LIN {X 0,Y 490.653,Z 372.898,A -85,B 0,C 180,E1 -6548.135,E2 -6548.135} C_VEL
LIN {X 0,Y 489.787,Z 400.79,A -85,B 0,C 180,E1 -6551.814,E2 -6551.814} C_VEL
LIN {X 0,Y 489.394,Z 415.444,A -85,B 0,C 180,E1 -6553.727,E2 -6553.727} C_VEL
LIN {X 0,Y 491.542,Z 434.875,A -85,B 0,C 180,E1 -6554.12,E2 -6554.12} C_VEL
LIN {X 0,Y 490.743,Z 525.863,A -85,B 0,C 180,E1 -6555.565,E2 -6555.565} C_VEL
LIN {X 0,Y 490.418,Z 538.788,A -85,B 0,C 180,E1 -6555.926,E2 -6555.926} C_VEL
LIN {X 0,Y 490.051,Z 550.862,A -85,B 0,C 180,E1 -6556.418,E2 -6556.418} C_VEL
LIN {X 0,Y 489.656,Z 562.336,A -85,B 0,C 180,E1 -6557.04,E2 -6557.04} C_VEL
LIN {X 0,Y 489.306,Z 574.419,A -85,B 0,C 180,E1 -6557.892,E2 -6557.892} C_VEL
LIN {X 0,Y 488.89,Z 584.844,A -85,B 0,C 180,E1 -6558.809,E2 -6558.809} C_VEL
LIN {X 0,Y 488.611,Z 594.472,A -85,B 0,C 180,E1 -6559.851,E2 -6559.851} C_VEL
LIN {X 0,Y 488.372,Z 603.748,A -85,B 0,C 180,E1 -6561.1,E2 -6561.1} C_VEL
LIN {X 0,Y 488.223,Z 611.226,A -85,B 0,C 180,E1 -6562.348,E2 -6562.348} C_VEL
LIN {X 0,Y 488.085,Z 617.817,A -85,B 0,C 180,E1 -6563.74,E2 -6563.74} C_VEL
LIN {X 0,Y 488.036,Z 622.557,A -85,B 0,C 180,E1 -6565.043,E2 -6565.043} C_VEL
LIN {X 0,Y 488.119,Z 624.938,A -85,B 0,C 180,E1 -6565.872,E2 -6565.872} C_VEL
LIN {X 0,Y 488.124,Z 626.864,A -85,B 0,C 180,E1 -6566.698,E2 -6566.698} C_VEL
LIN {X 0,Y 488.054,Z 628.303,A -85,B 0,C 180,E1 -6567.524,E2 -6567.524} C_VEL
LIN {X 0,Y 488.022,Z 629.312,A -85,B 0,C 180,E1 -6568.349,E2 -6568.349} C_VEL
LIN {X 0,Y 488.018,Z 629.915,A -85,B 0,C 180,E1 -6569.175,E2 -6569.175} C_VEL
LIN {X 0,Y 488.029,Z 630.112,A -85,B 0,C 180,E1 -6570,E2 -6570} C_VEL
LIN {X 0,Y 488.024,Z 629.858,A -85,B 0,C 180,E1 -6570.825,E2 -6570.825} C_VEL
LIN {X 0,Y 488.036,Z 629.184,A -85,B 0,C 180,E1 -6571.65,E2 -6571.65} C_VEL
LIN {X 0,Y 488.072,Z 628.103,A -85,B 0,C 180,E1 -6572.476,E2 -6572.476} C_VEL
LIN {X 0,Y 488.128,Z 626.599,A -85,B 0,C 180,E1 -6573.301,E2 -6573.301} C_VEL
LIN {X 0,Y 488.126,Z 623.454,A -85,B 0,C 180,E1 -6574.542,E2 -6574.542} C_VEL
LIN {X 0,Y 488.195,Z 618.077,A -85,B 0,C 180,E1 -6576.063,E2 -6576.063} C_VEL
LIN {X 0,Y 488.22,Z 611.62,A -85,B 0,C 180,E1 -6577.444,E2 -6577.444} C_VEL
LIN {X 0,Y 488.343,Z 604.254,A -85,B 0,C 180,E1 -6578.691,E2 -6578.691} C_VEL
LIN {X 0,Y 488.562,Z 595.04,A -85,B 0,C 180,E1 -6579.94,E2 -6579.94} C_VEL
LIN {X 0,Y 488.865,Z 585.619,A -85,B 0,C 180,E1 -6580.981,E2 -6580.981} C_VEL
LIN {X 0,Y 489.197,Z 574.668,A -85,B 0,C 180,E1 -6581.962,E2 -6581.962} C_VEL
LIN {X 0,Y 489.551,Z 563.67,A -85,B 0,C 180,E1 -6582.751,E2 -6582.751} C_VEL
LIN {X 0,Y 489.887,Z 551.761,A -85,B 0,C 180,E1 -6583.428,E2 -6583.428} C_VEL
LIN {X 0,Y 490.278,Z 538.993,A -85,B 0,C 180,E1 -6583.972,E2 -6583.972} C_VEL
LIN {X 0,Y 490.602,Z 525.693,A -85,B 0,C 180,E1 -6584.36,E2 -6584.36} C_VEL
LIN {X 0,Y 490.844,Z 499.198,A -85,B 0,C 180,E1 -6584.803,E2 -6584.803} C_VEL
LIN {X 0,Y 491.269,Z 432.405,A -85,B 0,C 180,E1 -6585.878,E2 -6585.878} C_VEL
LIN {X 0,Y 489.151,Z 412.344,A -85,B 0,C 180,E1 -6586.298,E2 -6586.298} C_VEL
LIN {X 0,Y 489.707,Z 390.705,A -85,B 0,C 180,E1 -6589.093,E2 -6589.093} C_VEL
LIN {X 0,Y 490.304,Z 367.801,A -85,B 0,C 180,E1 -6592.103,E2 -6592.103} C_VEL
LIN {X 0,Y 491.003,Z 346.439,A -85,B 0,C 180,E1 -6594.977,E2 -6594.977} C_VEL
LIN {X 0,Y 491.359,Z 333.411,A -85,B 0,C 180,E1 -6596.779,E2 -6596.779} C_VEL
LIN {X 0,Y 488.723,Z 320.611,A -85,B 0,C 180,E1 -6598.777,E2 -6598.777} C_VEL
LIN {X 0,Y 488.706,Z 320.614,A -85,B 0,C 180,E1 -6601.954,E2 -6601.954} C_VEL
LIN {X 0,Y 488.722,Z 320.608,A -85,B 0,C 180,E1 -6604.947,E2 -6604.947} C_VEL
LIN {X 0,Y 488.677,Z 320.616,A -85,B 0,C 180,E1 -6608.2,E2 -6608.2} C_VEL
LIN {X 0,Y 488.695,Z 320.615,A -85,B 0,C 180,E1 -6610.341,E2 -6610.341} C_VEL
LIN {X 0,Y 488.677,Z 320.614,A -85,B 0,C 180,E1 -6613.656,E2 -6613.656} C_VEL
LIN {X 0,Y 488.677,Z 320.615,A -85,B 0,C 180,E1 -6616.344,E2 -6616.344} C_VEL
LIN {X 0,Y 488.706,Z 320.61,A -85,B 0,C 180,E1 -6619.673,E2 -6619.673} C_VEL
LIN {X 0,Y 488.651,Z 320.613,A -85,B 0,C 180,E1 -6622.838,E2 -6622.838} C_VEL
LIN {X 0,Y 488.719,Z 320.61,A -85,B 0,C 180,E1 -6625.886,E2 -6625.886} C_VEL
LIN {X 0,Y 488.684,Z 320.61,A -85,B 0,C 180,E1 -6628.819,E2 -6628.819} C_VEL
LIN {X 0,Y 488.693,Z 320.614,A -85,B 0,C 180,E1 -6631.668,E2 -6631.668} C_VEL
LIN {X 0,Y 488.695,Z 320.61,A -85,B 0,C 180,E1 -6634.961,E2 -6634.961} C_VEL
LIN {X 0,Y 488.684,Z 320.614,A -85,B 0,C 180,E1 -6638.042,E2 -6638.042} C_VEL
LIN {X 0,Y 488.709,Z 320.608,A -85,B 0,C 180,E1 -6640.685,E2 -6640.685} C_VEL
LIN {X 0,Y 488.756,Z 320.605,A -85,B 0,C 180,E1 -6644.144,E2 -6644.144} C_VEL
LIN {X 0,Y 488.736,Z 320.61,A -85,B 0,C 180,E1 -6646.077,E2 -6646.077} C_VEL
LIN {X 0,Y 491.729,Z 329.522,A -85,B 0,C 180,E1 -6646.349,E2 -6646.349} C_VEL
LIN {X 0,Y 490.884,Z 411.162,A -85,B 0,C 180,E1 -6647.703,E2 -6647.703} C_VEL
LIN {X 0,Y 490.845,Z 424.387,A -85,B 0,C 180,E1 -6648.096,E2 -6648.096} C_VEL
LIN {X 0,Y 490.644,Z 436.99,A -85,B 0,C 180,E1 -6648.641,E2 -6648.641} C_VEL
LIN {X 0,Y 490.383,Z 449.309,A -85,B 0,C 180,E1 -6649.366,E2 -6649.366} C_VEL
LIN {X 0,Y 490.036,Z 460.307,A -85,B 0,C 180,E1 -6650.194,E2 -6650.194} C_VEL
LIN {X 0,Y 489.745,Z 470.169,A -85,B 0,C 180,E1 -6651.125,E2 -6651.125} C_VEL
LIN {X 0,Y 489.407,Z 479.39,A -85,B 0,C 180,E1 -6652.2,E2 -6652.2} C_VEL
LIN {X 0,Y 489.033,Z 487.732,A -85,B 0,C 180,E1 -6653.398,E2 -6653.398} C_VEL
LIN {X 0,Y 488.876,Z 494.611,A -85,B 0,C 180,E1 -6654.638,E2 -6654.638} C_VEL
LIN {X 0,Y 488.585,Z 500.097,A -85,B 0,C 180,E1 -6655.875,E2 -6655.875} C_VEL
LIN {X 0,Y 488.461,Z 504.372,A -85,B 0,C 180,E1 -6657.113,E2 -6657.113} C_VEL
LIN {X 0,Y 488.395,Z 507.572,A -85,B 0,C 180,E1 -6658.35,E2 -6658.35} C_VEL
LIN {X 0,Y 488.302,Z 509.151,A -85,B 0,C 180,E1 -6659.175,E2 -6659.175} C_VEL
LIN {X 0,Y 488.274,Z 510.323,A -85,B 0,C 180,E1 -6660,E2 -6660} C_VEL
LIN {X 0,Y 488.28,Z 511.074,A -85,B 0,C 180,E1 -6660.824,E2 -6660.824} C_VEL
LIN {X 0,Y 488.145,Z 511.418,A -85,B 0,C 180,E1 -6661.65,E2 -6661.65} C_VEL
LIN {X 0,Y 488.243,Z 510.907,A -85,B 0,C 180,E1 -6663.3,E2 -6663.3} C_VEL
LIN {X 0,Y 488.28,Z 510.038,A -85,B 0,C 180,E1 -6664.127,E2 -6664.127} C_VEL
LIN {X 0,Y 488.292,Z 508.754,A -85,B 0,C 180,E1 -6664.954,E2 -6664.954} C_VEL
LIN {X 0,Y 488.415,Z 506.04,A -85,B 0,C 180,E1 -6666.195,E2 -6666.195} C_VEL
LIN {X 0,Y 488.535,Z 502.302,A -85,B 0,C 180,E1 -6667.439,E2 -6667.439} C_VEL
LIN {X 0,Y 488.653,Z 497.43,A -85,B 0,C 180,E1 -6668.685,E2 -6668.685} C_VEL
LIN {X 0,Y 488.843,Z 491.265,A -85,B 0,C 180,E1 -6669.934,E2 -6669.934} C_VEL
LIN {X 0,Y 489.121,Z 483.572,A -85,B 0,C 180,E1 -6671.185,E2 -6671.185} C_VEL
LIN {X 0,Y 489.359,Z 475.615,A -85,B 0,C 180,E1 -6672.235,E2 -6672.235} C_VEL
LIN {X 0,Y 489.707,Z 465.965,A -85,B 0,C 180,E1 -6673.274,E2 -6673.274} C_VEL
LIN {X 0,Y 490.05,Z 455.168,A -85,B 0,C 180,E1 -6674.217,E2 -6674.217} C_VEL
LIN {X 0,Y 490.374,Z 444.676,A -85,B 0,C 180,E1 -6674.949,E2 -6674.949} C_VEL
LIN {X 0,Y 490.66,Z 432.035,A -85,B 0,C 180,E1 -6675.632,E2 -6675.632} C_VEL
LIN {X 0,Y 490.858,Z 418.426,A -85,B 0,C 180,E1 -6676.167,E2 -6676.167} C_VEL
LIN {X 0,Y 490.986,Z 405.659,A -85,B 0,C 180,E1 -6676.488,E2 -6676.488} C_VEL
LIN {X 0,Y 491.581,Z 329.224,A -85,B 0,C 180,E1 -6677.701,E2 -6677.701} C_VEL
LIN {X 0,Y 488.75,Z 320.604,A -85,B 0,C 180,E1 -6677.95,E2 -6677.95} C_VEL
LIN {X 0,Y 488.708,Z 320.609,A -85,B 0,C 180,E1 -6681.07,E2 -6681.07} C_VEL
LIN {X 0,Y 488.689,Z 320.608,A -85,B 0,C 180,E1 -6683.745,E2 -6683.745} C_VEL
LIN {X 0,Y 488.792,Z 320.599,A -85,B 0,C 180,E1 -6686.943,E2 -6686.943} C_VEL
LIN {X 0,Y 488.709,Z 320.61,A -85,B 0,C 180,E1 -6690.362,E2 -6690.362} C_VEL
LIN {X 0,Y 488.729,Z 320.603,A -85,B 0,C 180,E1 -6693.483,E2 -6693.483} C_VEL
LIN {X 0,Y 488.682,Z 320.613,A -85,B 0,C 180,E1 -6696.354,E2 -6696.354} C_VEL
LIN {X 0,Y 488.7,Z 320.607,A -85,B 0,C 180,E1 -6699.254,E2 -6699.254} C_VEL
LIN {X 0,Y 488.706,Z 320.606,A -85,B 0,C 180,E1 -6701.599,E2 -6701.599} C_VEL
LIN {X 0,Y 488.7,Z 320.61,A -85,B 0,C 180,E1 -6704.802,E2 -6704.802} C_VEL
LIN {X 0,Y 488.69,Z 320.608,A -85,B 0,C 180,E1 -6707.474,E2 -6707.474} C_VEL
LIN {X 0,Y 488.731,Z 320.603,A -85,B 0,C 180,E1 -6709.676,E2 -6709.676} C_VEL
LIN {X 0,Y 488.673,Z 320.613,A -85,B 0,C 180,E1 -6712.523,E2 -6712.523} C_VEL
LIN {X 0,Y 488.011,Z 320.695,A -85,B 0,C 180,E1 -6713.211,E2 -6713.211} C_VEL
LIN {X 0,Y 485.159,Z 321.054,A -85,B 0,C 180,E1 -6714.329,E2 -6714.329} C_VEL
LIN {X 0,Y 482.762,Z 321.348,A -85,B 0,C 180,E1 -6715.23,E2 -6715.23} C_VEL
LIN {X 0,Y 481.756,Z 321.474,A -85,B 0,C 180,E1 -6715.926,E2 -6715.926} C_VEL
LIN {X 0,Y 481.688,Z 321.484,A -85,B 0,C 180,E1 -6716.162,E2 -6716.162} C_VEL
LIN {X 0,Y 481.648,Z 321.485,A -85,B 0,C 180,E1 -6719.417,E2 -6719.417} C_VEL
LIN {X 0,Y 481.698,Z 321.484,A -85,B 0,C 180,E1 -6722.168,E2 -6722.168} C_VEL
LIN {X 0,Y 481.716,Z 321.478,A -85,B 0,C 180,E1 -6724.97,E2 -6724.97} C_VEL
LIN {X 0,Y 481.648,Z 321.487,A -85,B 0,C 180,E1 -6727.705,E2 -6727.705} C_VEL
LIN {X 0,Y 481.703,Z 321.484,A -85,B 0,C 180,E1 -6730.393,E2 -6730.393} C_VEL
LIN {X 0,Y 481.688,Z 321.481,A -85,B 0,C 180,E1 -6733.034,E2 -6733.034} C_VEL
LIN {X 0,Y 481.687,Z 321.483,A -85,B 0,C 180,E1 -6735.639,E2 -6735.639} C_VEL
LIN {X 0,Y 481.748,Z 321.48,A -85,B 0,C 180,E1 -6738.215,E2 -6738.215} C_VEL
LIN {X 0,Y 481.76,Z 321.474,A -85,B 0,C 180,E1 -6741.612,E2 -6741.612} C_VEL
LIN {X 0,Y 481.814,Z 321.471,A -85,B 0,C 180,E1 -6744.14,E2 -6744.14} C_VEL
LIN {X 0,Y 481.926,Z 321.453,A -85,B 0,C 180,E1 -6747.493,E2 -6747.493} C_VEL
LIN {X 0,Y 481.903,Z 321.454,A -85,B 0,C 180,E1 -6750.836,E2 -6750.836} C_VEL
LIN {X 0,Y 481.926,Z 321.453,A -85,B 0,C 180,E1 -6752.508,E2 -6752.508} C_VEL
LIN {X 0,Y 481.814,Z 321.469,A -85,B 0,C 180,E1 -6755.861,E2 -6755.861} C_VEL
LIN {X 0,Y 481.76,Z 321.474,A -85,B 0,C 180,E1 -6758.389,E2 -6758.389} C_VEL
LIN {X 0,Y 481.749,Z 321.477,A -85,B 0,C 180,E1 -6761.785,E2 -6761.785} C_VEL
LIN {X 0,Y 481.741,Z 321.475,A -85,B 0,C 180,E1 -6765.225,E2 -6765.225} C_VEL
LIN {X 0,Y 481.71,Z 321.478,A -85,B 0,C 180,E1 -6768.722,E2 -6768.722} C_VEL
LIN {X 0,Y 481.645,Z 321.489,A -85,B 0,C 180,E1 -6771.395,E2 -6771.395} C_VEL
LIN {X 0,Y 481.676,Z 321.486,A -85,B 0,C 180,E1 -6774.113,E2 -6774.113} C_VEL
LIN {X 0,Y 481.746,Z 321.475,A -85,B 0,C 180,E1 -6777.14,E2 -6777.14} C_VEL
LIN {X 0,Y 481.678,Z 321.487,A -85,B 0,C 180,E1 -6779.742,E2 -6779.742} C_VEL
LIN {X 0,Y 481.672,Z 321.483,A -85,B 0,C 180,E1 -6782.675,E2 -6782.675} C_VEL
LIN {X 0,Y 481.641,Z 321.492,A -85,B 0,C 180,E1 -6785.71,E2 -6785.71} C_VEL
LIN {X 0,Y 481.671,Z 321.483,A -85,B 0,C 180,E1 -6788.86,E2 -6788.86} C_VEL
LIN {X 0,Y 481.652,Z 321.49,A -85,B 0,C 180,E1 -6791.913,E2 -6791.913} C_VEL
LIN {X 0,Y 481.655,Z 321.485,A -85,B 0,C 180,E1 -6794.459,E2 -6794.459} C_VEL
LIN {X 0,Y 481.648,Z 321.49,A -85,B 0,C 180,E1 -6797.84,E2 -6797.84} C_VEL
LIN {X 0,Y 481.662,Z 321.484,A -85,B 0,C 180,E1 -6800.655,E2 -6800.655} C_VEL
LIN {X 0,Y 481.629,Z 321.492,A -85,B 0,C 180,E1 -6803.377,E2 -6803.377} C_VEL
LIN {X 0,Y 481.678,Z 321.482,A -85,B 0,C 180,E1 -6806.328,E2 -6806.328} C_VEL
LIN {X 0,Y 481.652,Z 321.49,A -85,B 0,C 180,E1 -6809.418,E2 -6809.418} C_VEL
LIN {X 0,Y 481.702,Z 321.48,A -85,B 0,C 180,E1 -6812.169,E2 -6812.169} C_VEL
LIN {X 0,Y 481.715,Z 321.48,A -85,B 0,C 180,E1 -6814.97,E2 -6814.97} C_VEL
LIN {X 0,Y 481.696,Z 321.483,A -85,B 0,C 180,E1 -6815.913,E2 -6815.913} C_VEL
LIN {X 0,Y 484.725,Z 330.592,A -85,B 0,C 180,E1 -6816.19,E2 -6816.19} C_VEL
LIN {X 0,Y 484.061,Z 408.884,A -85,B 0,C 180,E1 -6817.457,E2 -6817.457} C_VEL
LIN {X 0,Y 483.915,Z 421.637,A -85,B 0,C 180,E1 -6817.815,E2 -6817.815} C_VEL
LIN {X 0,Y 483.75,Z 433.868,A -85,B 0,C 180,E1 -6818.326,E2 -6818.326} C_VEL
LIN {X 0,Y 483.457,Z 446.293,A -85,B 0,C 180,E1 -6819.025,E2 -6819.025} C_VEL
LIN {X 0,Y 483.096,Z 456.914,A -85,B 0,C 180,E1 -6819.787,E2 -6819.787} C_VEL
LIN {X 0,Y 482.759,Z 467.753,A -85,B 0,C 180,E1 -6820.77,E2 -6820.77} C_VEL
LIN {X 0,Y 482.412,Z 476.559,A -85,B 0,C 180,E1 -6821.747,E2 -6821.747} C_VEL
LIN {X 0,Y 482.1,Z 484.622,A -85,B 0,C 180,E1 -6822.831,E2 -6822.831} C_VEL
LIN {X 0,Y 481.854,Z 491.253,A -85,B 0,C 180,E1 -6823.912,E2 -6823.912} C_VEL
LIN {X 0,Y 481.621,Z 497.7,A -85,B 0,C 180,E1 -6825.205,E2 -6825.205} C_VEL
LIN {X 0,Y 481.43,Z 502.757,A -85,B 0,C 180,E1 -6826.493,E2 -6826.493} C_VEL
LIN {X 0,Y 481.375,Z 507.213,A -85,B 0,C 180,E1 -6828.014,E2 -6828.014} C_VEL
LIN {X 0,Y 481.26,Z 509.417,A -85,B 0,C 180,E1 -6829.057,E2 -6829.057} C_VEL
LIN {X 0,Y 481.183,Z 510.736,A -85,B 0,C 180,E1 -6829.906,E2 -6829.906} C_VEL
LIN {X 0,Y 481.219,Z 511.633,A -85,B 0,C 180,E1 -6830.756,E2 -6830.756} C_VEL
LIN {X 0,Y 481.205,Z 512.089,A -85,B 0,C 180,E1 -6831.602,E2 -6831.602} C_VEL
LIN {X 0,Y 481.297,Z 511.861,A -85,B 0,C 180,E1 -6833.197,E2 -6833.197} C_VEL
LIN {X 0,Y 481.291,Z 511.047,A -85,B 0,C 180,E1 -6834.134,E2 -6834.134} C_VEL
LIN {X 0,Y 481.355,Z 509.867,A -85,B 0,C 180,E1 -6834.975,E2 -6834.975} C_VEL
LIN {X 0,Y 481.394,Z 507.324,A -85,B 0,C 180,E1 -6836.234,E2 -6836.234} C_VEL
LIN {X 0,Y 481.518,Z 503.762,A -85,B 0,C 180,E1 -6837.491,E2 -6837.491} C_VEL
LIN {X 0,Y 481.668,Z 499.092,A -85,B 0,C 180,E1 -6838.746,E2 -6838.746} C_VEL
LIN {X 0,Y 481.926,Z 493.165,A -85,B 0,C 180,E1 -6840,E2 -6840} C_VEL
LIN {X 0,Y 482.206,Z 485.737,A -85,B 0,C 180,E1 -6841.253,E2 -6841.253} C_VEL
LIN {X 0,Y 482.601,Z 476.463,A -85,B 0,C 180,E1 -6842.504,E2 -6842.504} C_VEL
LIN {X 0,Y 482.949,Z 466.853,A -85,B 0,C 180,E1 -6843.546,E2 -6843.546} C_VEL
LIN {X 0,Y 483.238,Z 456.096,A -85,B 0,C 180,E1 -6844.484,E2 -6844.484} C_VEL
LIN {X 0,Y 483.609,Z 445.598,A -85,B 0,C 180,E1 -6845.212,E2 -6845.212} C_VEL
LIN {X 0,Y 483.863,Z 434.096,A -85,B 0,C 180,E1 -6845.836,E2 -6845.836} C_VEL
LIN {X 0,Y 484.003,Z 420.929,A -85,B 0,C 180,E1 -6846.357,E2 -6846.357} C_VEL
LIN {X 0,Y 484.123,Z 407.732,A -85,B 0,C 180,E1 -6846.696,E2 -6846.696} C_VEL
LIN {X 0,Y 484.791,Z 330.376,A -85,B 0,C 180,E1 -6847.974,E2 -6847.974} C_VEL
LIN {X 0,Y 481.72,Z 321.482,A -85,B 0,C 180,E1 -6848.265,E2 -6848.265} C_VEL
LIN {X 0,Y 481.728,Z 321.479,A -85,B 0,C 180,E1 -6851.786,E2 -6851.786} C_VEL
LIN {X 0,Y 481.742,Z 321.476,A -85,B 0,C 180,E1 -6855.225,E2 -6855.225} C_VEL
LIN {X 0,Y 481.645,Z 321.493,A -85,B 0,C 180,E1 -6858.725,E2 -6858.725} C_VEL
LIN {X 0,Y 481.625,Z 321.491,A -85,B 0,C 180,E1 -6861.396,E2 -6861.396} C_VEL
LIN {X 0,Y 481.646,Z 321.492,A -85,B 0,C 180,E1 -6864.115,E2 -6864.115} C_VEL
LIN {X 0,Y 481.646,Z 321.487,A -85,B 0,C 180,E1 -6867.115,E2 -6867.115} C_VEL
LIN {X 0,Y 481.66,Z 321.487,A -85,B 0,C 180,E1 -6869.743,E2 -6869.743} C_VEL
LIN {X 0,Y 481.656,Z 321.486,A -85,B 0,C 180,E1 -6872.676,E2 -6872.676} C_VEL
LIN {X 0,Y 481.653,Z 321.483,A -85,B 0,C 180,E1 -6875.202,E2 -6875.202} C_VEL
LIN {X 0,Y 481.634,Z 321.491,A -85,B 0,C 180,E1 -6878.003,E2 -6878.003} C_VEL
LIN {X 0,Y 481.627,Z 321.486,A -85,B 0,C 180,E1 -6881.045,E2 -6881.045} C_VEL
LIN {X 0,Y 481.658,Z 321.485,A -85,B 0,C 180,E1 -6884.458,E2 -6884.458} C_VEL
LIN {X 0,Y 481.633,Z 321.495,A -85,B 0,C 180,E1 -6887.837,E2 -6887.837} C_VEL
LIN {X 0,Y 481.669,Z 321.485,A -85,B 0,C 180,E1 -6891.14,E2 -6891.14} C_VEL
LIN {X 0,Y 481.661,Z 321.485,A -85,B 0,C 180,E1 -6894.797,E2 -6894.797} C_VEL
LIN {X 0,Y 481.66,Z 321.489,A -85,B 0,C 180,E1 -6897.811,E2 -6897.811} C_VEL
LIN {X 0,Y 481.736,Z 321.634,A -85,B 0,C 180,E1 -6900.659,E2 -6900.659} C_VEL
LIN {X 0,Y 484.857,Z 335.891,A -85,B 0,C 180,E1 -6902.832,E2 -6902.832} C_VEL
LIN {X 0,Y 484.986,Z 340.7,A -85,B 0,C 180,E1 -6903.511,E2 -6903.511} C_VEL
LIN {X 0,Y 484.028,Z 364.108,A -85,B 0,C 180,E1 -6906.712,E2 -6906.712} C_VEL
LIN {X 0,Y 483.302,Z 383.679,A -85,B 0,C 180,E1 -6909.351,E2 -6909.351} C_VEL
LIN {X 0,Y 482.633,Z 404.958,A -85,B 0,C 180,E1 -6912.194,E2 -6912.194} C_VEL
LIN {X 0,Y 482.405,Z 415.085,A -85,B 0,C 180,E1 -6913.501,E2 -6913.501} C_VEL
LIN {X 0,Y 484.667,Z 435.54,A -85,B 0,C 180,E1 -6913.918,E2 -6913.918} C_VEL
LIN {X 0,Y 483.827,Z 525.311,A -85,B 0,C 180,E1 -6915.381,E2 -6915.381} C_VEL
LIN {X 0,Y 483.44,Z 538.896,A -85,B 0,C 180,E1 -6915.772,E2 -6915.772} C_VEL
LIN {X 0,Y 483.036,Z 551.808,A -85,B 0,C 180,E1 -6916.324,E2 -6916.324} C_VEL
LIN {X 0,Y 482.616,Z 562.838,A -85,B 0,C 180,E1 -6916.955,E2 -6916.955} C_VEL
LIN {X 0,Y 482.262,Z 574.328,A -85,B 0,C 180,E1 -6917.791,E2 -6917.791} C_VEL
LIN {X 0,Y 481.809,Z 584.929,A -85,B 0,C 180,E1 -6918.749,E2 -6918.749} C_VEL
LIN {X 0,Y 481.565,Z 593.523,A -85,B 0,C 180,E1 -6919.701,E2 -6919.701} C_VEL
LIN {X 0,Y 481.312,Z 602.832,A -85,B 0,C 180,E1 -6920.969,E2 -6920.969} C_VEL
LIN {X 0,Y 481.142,Z 610.331,A -85,B 0,C 180,E1 -6922.235,E2 -6922.235} C_VEL
LIN {X 0,Y 481.078,Z 615.98,A -85,B 0,C 180,E1 -6923.417,E2 -6923.417} C_VEL
LIN {X 0,Y 481.019,Z 620.328,A -85,B 0,C 180,E1 -6924.55,E2 -6924.55} C_VEL
LIN {X 0,Y 481.059,Z 624.088,A -85,B 0,C 180,E1 -6925.811,E2 -6925.811} C_VEL
LIN {X 0,Y 481.073,Z 626.018,A -85,B 0,C 180,E1 -6926.65,E2 -6926.65} C_VEL
LIN {X 0,Y 480.998,Z 627.46,A -85,B 0,C 180,E1 -6927.488,E2 -6927.488} C_VEL
LIN {X 0,Y 480.968,Z 628.467,A -85,B 0,C 180,E1 -6928.325,E2 -6928.325} C_VEL
LIN {X 0,Y 480.966,Z 629.069,A -85,B 0,C 180,E1 -6929.163,E2 -6929.163} C_VEL
LIN {X 0,Y 480.981,Z 629.262,A -85,B 0,C 180,E1 -6930,E2 -6930} C_VEL
LIN {X 0,Y 480.975,Z 628.997,A -85,B 0,C 180,E1 -6930.837,E2 -6930.837} C_VEL
LIN {X 0,Y 480.985,Z 628.313,A -85,B 0,C 180,E1 -6931.674,E2 -6931.674} C_VEL
LIN {X 0,Y 481.019,Z 627.222,A -85,B 0,C 180,E1 -6932.512,E2 -6932.512} C_VEL
LIN {X 0,Y 481.078,Z 624.745,A -85,B 0,C 180,E1 -6933.769,E2 -6933.769} C_VEL
LIN {X 0,Y 481.039,Z 621.208,A -85,B 0,C 180,E1 -6935.029,E2 -6935.029} C_VEL
LIN {X 0,Y 481.121,Z 616.306,A -85,B 0,C 180,E1 -6936.35,E2 -6936.35} C_VEL
LIN {X 0,Y 481.181,Z 609.489,A -85,B 0,C 180,E1 -6937.764,E2 -6937.764} C_VEL
LIN {X 0,Y 481.313,Z 601.779,A -85,B 0,C 180,E1 -6939.031,E2 -6939.031} C_VEL
LIN {X 0,Y 481.559,Z 592.216,A -85,B 0,C 180,E1 -6940.299,E2 -6940.299} C_VEL
LIN {X 0,Y 481.819,Z 582.279,A -85,B 0,C 180,E1 -6941.357,E2 -6941.357} C_VEL
LIN {X 0,Y 482.174,Z 571.65,A -85,B 0,C 180,E1 -6942.28,E2 -6942.28} C_VEL
LIN {X 0,Y 482.584,Z 560.752,A -85,B 0,C 180,E1 -6943.046,E2 -6943.046} C_VEL
LIN {X 0,Y 482.961,Z 548.243,A -85,B 0,C 180,E1 -6943.732,E2 -6943.732} C_VEL
LIN {X 0,Y 483.417,Z 534.462,A -85,B 0,C 180,E1 -6944.282,E2 -6944.282} C_VEL
LIN {X 0,Y 483.793,Z 521.74,A -85,B 0,C 180,E1 -6944.62,E2 -6944.62} C_VEL
LIN {X 0,Y 484.493,Z 433.696,A -85,B 0,C 180,E1 -6946.075,E2 -6946.075} C_VEL
LIN {X 0,Y 482.144,Z 411.17,A -85,B 0,C 180,E1 -6946.568,E2 -6946.568} C_VEL
LIN {X 0,Y 482.642,Z 390.052,A -85,B 0,C 180,E1 -6949.348,E2 -6949.348} C_VEL
LIN {X 0,Y 483.337,Z 368.644,A -85,B 0,C 180,E1 -6952.213,E2 -6952.213} C_VEL
LIN {X 0,Y 484.083,Z 347.416,A -85,B 0,C 180,E1 -6955.129,E2 -6955.129} C_VEL
LIN {X 0,Y 484.459,Z 334.635,A -85,B 0,C 180,E1 -6956.942,E2 -6956.942} C_VEL
LIN {X 0,Y 481.694,Z 321.486,A -85,B 0,C 180,E1 -6959.05,E2 -6959.05} C_VEL
LIN {X 0,Y 481.659,Z 321.493,A -85,B 0,C 180,E1 -6962.189,E2 -6962.189} C_VEL
LIN {X 0,Y 481.661,Z 321.486,A -85,B 0,C 180,E1 -6965.203,E2 -6965.203} C_VEL
LIN {X 0,Y 481.668,Z 321.487,A -85,B 0,C 180,E1 -6968.859,E2 -6968.859} C_VEL
LIN {X 0,Y 481.631,Z 321.495,A -85,B 0,C 180,E1 -6972.163,E2 -6972.163} C_VEL
LIN {X 0,Y 481.656,Z 321.487,A -85,B 0,C 180,E1 -6975.542,E2 -6975.542} C_VEL
LIN {X 0,Y 481.628,Z 321.489,A -85,B 0,C 180,E1 -6978.955,E2 -6978.955} C_VEL
LIN {X 0,Y 481.633,Z 321.492,A -85,B 0,C 180,E1 -6981.996,E2 -6981.996} C_VEL
LIN {X 0,Y 481.68,Z 321.483,A -85,B 0,C 180,E1 -6985.317,E2 -6985.317} C_VEL
LIN {X 0,Y 481.64,Z 321.49,A -85,B 0,C 180,E1 -6988.311,E2 -6988.311} C_VEL
LIN {X 0,Y 481.655,Z 321.487,A -85,B 0,C 180,E1 -6991.215,E2 -6991.215} C_VEL
LIN {X 0,Y 481.621,Z 321.495,A -85,B 0,C 180,E1 -6994.038,E2 -6994.038} C_VEL
LIN {X 0,Y 481.654,Z 321.488,A -85,B 0,C 180,E1 -6996.818,E2 -6996.818} C_VEL
LIN {X 0,Y 481.659,Z 321.492,A -85,B 0,C 180,E1 -6999.501,E2 -6999.501} C_VEL
LIN {X 0,Y 481.665,Z 321.487,A -85,B 0,C 180,E1 -7002.156,E2 -7002.156} C_VEL
LIN {X 0,Y 481.74,Z 321.48,A -85,B 0,C 180,E1 -7004.775,E2 -7004.775} C_VEL
LIN {X 0,Y 481.681,Z 321.49,A -85,B 0,C 180,E1 -7005.814,E2 -7005.814} C_VEL
LIN {X 0,Y 484.997,Z 331.124,A -85,B 0,C 180,E1 -7006.124,E2 -7006.124} C_VEL
LIN {X 0,Y 484.028,Z 411.924,A -85,B 0,C 180,E1 -7007.5,E2 -7007.5} C_VEL
LIN {X 0,Y 483.966,Z 425.906,A -85,B 0,C 180,E1 -7007.924,E2 -7007.924} C_VEL
LIN {X 0,Y 483.762,Z 438.322,A -85,B 0,C 180,E1 -7008.477,E2 -7008.477} C_VEL
LIN {X 0,Y 483.516,Z 450.549,A -85,B 0,C 180,E1 -7009.214,E2 -7009.214} C_VEL
LIN {X 0,Y 483.124,Z 461.485,A -85,B 0,C 180,E1 -7010.052,E2 -7010.052} C_VEL
LIN {X 0,Y 482.81,Z 471.288,A -85,B 0,C 180,E1 -7010.997,E2 -7010.997} C_VEL
LIN {X 0,Y 482.4,Z 481.13,A -85,B 0,C 180,E1 -7012.173,E2 -7012.173} C_VEL
LIN {X 0,Y 482.073,Z 488.785,A -85,B 0,C 180,E1 -7013.302,E2 -7013.302} C_VEL
LIN {X 0,Y 481.881,Z 495.639,A -85,B 0,C 180,E1 -7014.56,E2 -7014.56} C_VEL
LIN {X 0,Y 481.575,Z 501.101,A -85,B 0,C 180,E1 -7015.815,E2 -7015.815} C_VEL
LIN {X 0,Y 481.439,Z 505.35,A -85,B 0,C 180,E1 -7017.071,E2 -7017.071} C_VEL
LIN {X 0,Y 481.37,Z 508.522,A -85,B 0,C 180,E1 -7018.326,E2 -7018.326} C_VEL
LIN {X 0,Y 481.277,Z 510.086,A -85,B 0,C 180,E1 -7019.163,E2 -7019.163} C_VEL
LIN {X 0,Y 481.247,Z 511.242,A -85,B 0,C 180,E1 -7020,E2 -7020} C_VEL
LIN {X 0,Y 481.252,Z 511.965,A -85,B 0,C 180,E1 -7020.836,E2 -7020.836} C_VEL
LIN {X 0,Y 481.1,Z 512.292,A -85,B 0,C 180,E1 -7021.674,E2 -7021.674} C_VEL
LIN {X 0,Y 481.198,Z 511.739,A -85,B 0,C 180,E1 -7023.349,E2 -7023.349} C_VEL
LIN {X 0,Y 481.247,Z 510.834,A -85,B 0,C 180,E1 -7024.187,E2 -7024.187} C_VEL
LIN {X 0,Y 481.264,Z 509.523,A -85,B 0,C 180,E1 -7025.026,E2 -7025.026} C_VEL
LIN {X 0,Y 481.385,Z 506.761,A -85,B 0,C 180,E1 -7026.286,E2 -7026.286} C_VEL
LIN {X 0,Y 481.512,Z 502.968,A -85,B 0,C 180,E1 -7027.548,E2 -7027.548} C_VEL
LIN {X 0,Y 481.657,Z 498.032,A -85,B 0,C 180,E1 -7028.812,E2 -7028.812} C_VEL
LIN {X 0,Y 481.845,Z 491.8,A -85,B 0,C 180,E1 -7030.08,E2 -7030.08} C_VEL
LIN {X 0,Y 482.152,Z 484.004,A -85,B 0,C 180,E1 -7031.348,E2 -7031.348} C_VEL
LIN {X 0,Y 482.477,Z 474.449,A -85,B 0,C 180,E1 -7032.589,E2 -7032.589} C_VEL
LIN {X 0,Y 482.819,Z 463.975,A -85,B 0,C 180,E1 -7033.682,E2 -7033.682} C_VEL
LIN {X 0,Y 483.202,Z 452.363,A -85,B 0,C 180,E1 -7034.638,E2 -7034.638} C_VEL
LIN {X 0,Y 483.576,Z 440.934,A -85,B 0,C 180,E1 -7035.38,E2 -7035.38} C_VEL
LIN {X 0,Y 483.837,Z 429.194,A -85,B 0,C 180,E1 -7035.966,E2 -7035.966} C_VEL
LIN {X 0,Y 483.994,Z 415.59,A -85,B 0,C 180,E1 -7036.452,E2 -7036.452} C_VEL
LIN {X 0,Y 484.109,Z 402.044,A -85,B 0,C 180,E1 -7036.751,E2 -7036.751} C_VEL
LIN {X 0,Y 484.663,Z 330.407,A -85,B 0,C 180,E1 -7037.909,E2 -7037.909} C_VEL
LIN {X 0,Y 481.728,Z 321.48,A -85,B 0,C 180,E1 -7038.161,E2 -7038.161} C_VEL
LIN {X 0,Y 481.704,Z 321.483,A -85,B 0,C 180,E1 -7040.972,E2 -7040.972} C_VEL
LIN {X 0,Y 481.674,Z 321.484,A -85,B 0,C 180,E1 -7044.113,E2 -7044.113} C_VEL
LIN {X 0,Y 481.747,Z 321.475,A -85,B 0,C 180,E1 -7047.139,E2 -7047.139} C_VEL
LIN {X 0,Y 481.678,Z 321.482,A -85,B 0,C 180,E1 -7049.741,E2 -7049.741} C_VEL
LIN {X 0,Y 481.67,Z 321.49,A -85,B 0,C 180,E1 -7052.674,E2 -7052.674} C_VEL
LIN {X 0,Y 481.635,Z 321.487,A -85,B 0,C 180,E1 -7055.709,E2 -7055.709} C_VEL
LIN {X 0,Y 481.67,Z 321.486,A -85,B 0,C 180,E1 -7058.859,E2 -7058.859} C_VEL
LIN {X 0,Y 481.651,Z 321.486,A -85,B 0,C 180,E1 -7061.912,E2 -7061.912} C_VEL
LIN {X 0,Y 481.653,Z 321.491,A -85,B 0,C 180,E1 -7064.457,E2 -7064.457} C_VEL
LIN {X 0,Y 481.646,Z 321.487,A -85,B 0,C 180,E1 -7067.839,E2 -7067.839} C_VEL
LIN {X 0,Y 481.679,Z 321.486,A -85,B 0,C 180,E1 -7070.651,E2 -7070.651} C_VEL
LIN {X 0,Y 481.629,Z 321.488,A -85,B 0,C 180,E1 -7073.375,E2 -7073.375} C_VEL
LIN {X 0,Y 481.688,Z 321.484,A -85,B 0,C 180,E1 -7076.162,E2 -7076.162} C_VEL
LIN {X 0,Y 481.054,Z 321.57,A -85,B 0,C 180,E1 -7076.859,E2 -7076.859} C_VEL
LIN {X 0,Y 478.198,Z 321.927,A -85,B 0,C 180,E1 -7077.991,E2 -7077.991} C_VEL
LIN {X 0,Y 475.753,Z 322.227,A -85,B 0,C 180,E1 -7078.904,E2 -7078.904} C_VEL
LIN {X 0,Y 474.691,Z 322.355,A -85,B 0,C 180,E1 -7079.609,E2 -7079.609} C_VEL
LIN {X 0,Y 474.599,Z 322.365,A -85,B 0,C 180,E1 -7079.848,E2 -7079.848} C_VEL
LIN {X 0,Y 474.695,Z 322.355,A -85,B 0,C 180,E1 -7082.68,E2 -7082.68} C_VEL
LIN {X 0,Y 474.657,Z 322.357,A -85,B 0,C 180,E1 -7085.507,E2 -7085.507} C_VEL
LIN {X 0,Y 474.668,Z 322.355,A -85,B 0,C 180,E1 -7089.185,E2 -7089.185} C_VEL
LIN {X 0,Y 474.655,Z 322.359,A -85,B 0,C 180,E1 -7091.884,E2 -7091.884} C_VEL
LIN {X 0,Y 474.697,Z 322.355,A -85,B 0,C 180,E1 -7094.544,E2 -7094.544} C_VEL
LIN {X 0,Y 474.702,Z 322.355,A -85,B 0,C 180,E1 -7098.038,E2 -7098.038} C_VEL
LIN {X 0,Y 474.725,Z 322.349,A -85,B 0,C 180,E1 -7101.487,E2 -7101.487} C_VEL
LIN {X 0,Y 474.777,Z 322.347,A -85,B 0,C 180,E1 -7104.052,E2 -7104.052} C_VEL
LIN {X 0,Y 474.892,Z 322.329,A -85,B 0,C 180,E1 -7107.456,E2 -7107.456} C_VEL
LIN {X 0,Y 474.91,Z 322.33,A -85,B 0,C 180,E1 -7110,E2 -7110} C_VEL
LIN {X 0,Y 474.892,Z 322.329,A -85,B 0,C 180,E1 -7112.545,E2 -7112.545} C_VEL
LIN {X 0,Y 474.777,Z 322.347,A -85,B 0,C 180,E1 -7115.948,E2 -7115.948} C_VEL
LIN {X 0,Y 474.726,Z 322.35,A -85,B 0,C 180,E1 -7118.514,E2 -7118.514} C_VEL
LIN {X 0,Y 474.702,Z 322.357,A -85,B 0,C 180,E1 -7121.963,E2 -7121.963} C_VEL
LIN {X 0,Y 474.698,Z 322.354,A -85,B 0,C 180,E1 -7125.456,E2 -7125.456} C_VEL
LIN {X 0,Y 474.663,Z 322.356,A -85,B 0,C 180,E1 -7129.011,E2 -7129.011} C_VEL
LIN {X 0,Y 474.59,Z 322.369,A -85,B 0,C 180,E1 -7131.729,E2 -7131.729} C_VEL
LIN {X 0,Y 474.658,Z 322.357,A -85,B 0,C 180,E1 -7134.493,E2 -7134.493} C_VEL
LIN {X 0,Y 474.698,Z 322.354,A -85,B 0,C 180,E1 -7137.339,E2 -7137.339} C_VEL
LIN {X 0,Y 474.603,Z 322.363,A -85,B 0,C 180,E1 -7140.811,E2 -7140.811} C_VEL
LIN {X 0,Y 474.638,Z 322.364,A -85,B 0,C 180,E1 -7143.985,E2 -7143.985} C_VEL
LIN {X 0,Y 474.574,Z 322.368,A -85,B 0,C 180,E1 -7146.9,E2 -7146.9} C_VEL
LIN {X 0,Y 474.628,Z 322.365,A -85,B 0,C 180,E1 -7149.648,E2 -7149.648} C_VEL
LIN {X 0,Y 474.614,Z 322.363,A -85,B 0,C 180,E1 -7152.935,E2 -7152.935} C_VEL
LIN {X 0,Y 474.607,Z 322.367,A -85,B 0,C 180,E1 -7155.895,E2 -7155.895} C_VEL
LIN {X 0,Y 474.628,Z 322.363,A -85,B 0,C 180,E1 -7159.041,E2 -7159.041} C_VEL
LIN {X 0,Y 474.611,Z 322.368,A -85,B 0,C 180,E1 -7161.705,E2 -7161.705} C_VEL
LIN {X 0,Y 474.624,Z 322.361,A -85,B 0,C 180,E1 -7164.726,E2 -7164.726} C_VEL
LIN {X 0,Y 474.636,Z 322.363,A -85,B 0,C 180,E1 -7167.788,E2 -7167.788} C_VEL
LIN {X 0,Y 474.625,Z 322.363,A -85,B 0,C 180,E1 -7170.885,E2 -7170.885} C_VEL
LIN {X 0,Y 474.661,Z 322.36,A -85,B 0,C 180,E1 -7173.629,E2 -7173.629} C_VEL
LIN {X 0,Y 474.646,Z 322.363,A -85,B 0,C 180,E1 -7175.692,E2 -7175.692} C_VEL
LIN {X 0,Y 477.845,Z 331.959,A -85,B 0,C 180,E1 -7175.982,E2 -7175.982} C_VEL
LIN {X 0,Y 477.163,Z 410.39,A -85,B 0,C 180,E1 -7177.284,E2 -7177.284} C_VEL
LIN {X 0,Y 477.046,Z 422.813,A -85,B 0,C 180,E1 -7177.647,E2 -7177.647} C_VEL
LIN {X 0,Y 476.821,Z 435.905,A -85,B 0,C 180,E1 -7178.215,E2 -7178.215} C_VEL
LIN {X 0,Y 476.502,Z 448.176,A -85,B 0,C 180,E1 -7178.93,E2 -7178.93} C_VEL
LIN {X 0,Y 476.112,Z 459.837,A -85,B 0,C 180,E1 -7179.816,E2 -7179.816} C_VEL
LIN {X 0,Y 475.728,Z 470.304,A -85,B 0,C 180,E1 -7180.811,E2 -7180.811} C_VEL
LIN {X 0,Y 475.339,Z 479.662,A -85,B 0,C 180,E1 -7181.912,E2 -7181.912} C_VEL
LIN {X 0,Y 475,Z 488.679,A -85,B 0,C 180,E1 -7183.231,E2 -7183.231} C_VEL
LIN {X 0,Y 474.737,Z 495.84,A -85,B 0,C 180,E1 -7184.546,E2 -7184.546} C_VEL
LIN {X 0,Y 474.488,Z 501.491,A -85,B 0,C 180,E1 -7185.854,E2 -7185.854} C_VEL
LIN {X 0,Y 474.361,Z 505.882,A -85,B 0,C 180,E1 -7187.16,E2 -7187.16} C_VEL
LIN {X 0,Y 474.345,Z 508.189,A -85,B 0,C 180,E1 -7188.029,E2 -7188.029} C_VEL
LIN {X 0,Y 474.228,Z 510.016,A -85,B 0,C 180,E1 -7188.892,E2 -7188.892} C_VEL
LIN {X 0,Y 474.143,Z 511.397,A -85,B 0,C 180,E1 -7189.755,E2 -7189.755} C_VEL
LIN {X 0,Y 474.178,Z 512.364,A -85,B 0,C 180,E1 -7190.617,E2 -7190.617} C_VEL
LIN {X 0,Y 474.18,Z 512.902,A -85,B 0,C 180,E1 -7191.477,E2 -7191.477} C_VEL
LIN {X 0,Y 474.264,Z 512.734,A -85,B 0,C 180,E1 -7193.192,E2 -7193.192} C_VEL
LIN {X 0,Y 474.26,Z 512.057,A -85,B 0,C 180,E1 -7194.046,E2 -7194.046} C_VEL
LIN {X 0,Y 474.305,Z 510.927,A -85,B 0,C 180,E1 -7194.9,E2 -7194.9} C_VEL
LIN {X 0,Y 474.303,Z 509.408,A -85,B 0,C 180,E1 -7195.752,E2 -7195.752} C_VEL
LIN {X 0,Y 474.416,Z 506.293,A -85,B 0,C 180,E1 -7197.028,E2 -7197.028} C_VEL
LIN {X 0,Y 474.574,Z 502.117,A -85,B 0,C 180,E1 -7198.303,E2 -7198.303} C_VEL
LIN {X 0,Y 474.817,Z 496.756,A -85,B 0,C 180,E1 -7199.576,E2 -7199.576} C_VEL
LIN {X 0,Y 475.146,Z 489.988,A -85,B 0,C 180,E1 -7200.848,E2 -7200.848} C_VEL
LIN {X 0,Y 475.513,Z 481.565,A -85,B 0,C 180,E1 -7202.118,E2 -7202.118} C_VEL
LIN {X 0,Y 475.89,Z 472.919,A -85,B 0,C 180,E1 -7203.175,E2 -7203.175} C_VEL
LIN {X 0,Y 476.272,Z 463.355,A -85,B 0,C 180,E1 -7204.126,E2 -7204.126} C_VEL
LIN {X 0,Y 476.544,Z 452.883,A -85,B 0,C 180,E1 -7204.971,E2 -7204.971} C_VEL
LIN {X 0,Y 476.93,Z 441.262,A -85,B 0,C 180,E1 -7205.709,E2 -7205.709} C_VEL
LIN {X 0,Y 477.06,Z 429.199,A -85,B 0,C 180,E1 -7206.291,E2 -7206.291} C_VEL
LIN {X 0,Y 477.221,Z 415.862,A -85,B 0,C 180,E1 -7206.74,E2 -7206.74} C_VEL
LIN {X 0,Y 477.302,Z 401.245,A -85,B 0,C 180,E1 -7207.031,E2 -7207.031} C_VEL
LIN {X 0,Y 478.193,Z 332.453,A -85,B 0,C 180,E1 -7208.193,E2 -7208.193} C_VEL
LIN {X 0,Y 474.712,Z 322.574,A -85,B 0,C 180,E1 -7208.514,E2 -7208.514} C_VEL
LIN {X 0,Y 474.674,Z 322.362,A -85,B 0,C 180,E1 -7208.729,E2 -7208.729} C_VEL
LIN {X 0,Y 474.693,Z 322.359,A -85,B 0,C 180,E1 -7212.269,E2 -7212.269} C_VEL
LIN {X 0,Y 474.684,Z 322.356,A -85,B 0,C 180,E1 -7215.767,E2 -7215.767} C_VEL
LIN {X 0,Y 474.598,Z 322.369,A -85,B 0,C 180,E1 -7219.013,E2 -7219.013} C_VEL
LIN {X 0,Y 474.574,Z 322.371,A -85,B 0,C 180,E1 -7221.73,E2 -7221.73} C_VEL
LIN {X 0,Y 474.625,Z 322.367,A -85,B 0,C 180,E1 -7224.495,E2 -7224.495} C_VEL
LIN {X 0,Y 474.597,Z 322.365,A -85,B 0,C 180,E1 -7227.327,E2 -7227.327} C_VEL
LIN {X 0,Y 474.591,Z 322.37,A -85,B 0,C 180,E1 -7230.232,E2 -7230.232} C_VEL
LIN {X 0,Y 474.619,Z 322.361,A -85,B 0,C 180,E1 -7233.222,E2 -7233.222} C_VEL
LIN {X 0,Y 474.574,Z 322.369,A -85,B 0,C 180,E1 -7236.325,E2 -7236.325} C_VEL
LIN {X 0,Y 474.605,Z 322.365,A -85,B 0,C 180,E1 -7239.644,E2 -7239.644} C_VEL
LIN {X 0,Y 474.573,Z 322.365,A -85,B 0,C 180,E1 -7242.939,E2 -7242.939} C_VEL
LIN {X 0,Y 474.606,Z 322.368,A -85,B 0,C 180,E1 -7245.894,E2 -7245.894} C_VEL
LIN {X 0,Y 474.609,Z 322.363,A -85,B 0,C 180,E1 -7249.044,E2 -7249.044} C_VEL
LIN {X 0,Y 474.609,Z 322.368,A -85,B 0,C 180,E1 -7251.705,E2 -7251.705} C_VEL
LIN {X 0,Y 474.623,Z 322.361,A -85,B 0,C 180,E1 -7254.725,E2 -7254.725} C_VEL
LIN {X 0,Y 474.639,Z 322.364,A -85,B 0,C 180,E1 -7257.788,E2 -7257.788} C_VEL
LIN {X 0,Y 474.666,Z 322.422,A -85,B 0,C 180,E1 -7260.416,E2 -7260.416} C_VEL
LIN {X 0,Y 478.094,Z 338.449,A -85,B 0,C 180,E1 -7262.89,E2 -7262.89} C_VEL
LIN {X 0,Y 477.652,Z 351.673,A -85,B 0,C 180,E1 -7264.742,E2 -7264.742} C_VEL
LIN {X 0,Y 476.593,Z 377.996,A -85,B 0,C 180,E1 -7268.367,E2 -7268.367} C_VEL
LIN {X 0,Y 475.728,Z 402.575,A -85,B 0,C 180,E1 -7271.704,E2 -7271.704} C_VEL
LIN {X 0,Y 475.38,Z 414.058,A -85,B 0,C 180,E1 -7273.25,E2 -7273.25} C_VEL
LIN {X 0,Y 477.804,Z 436.037,A -85,B 0,C 180,E1 -7273.711,E2 -7273.711} C_VEL
LIN {X 0,Y 476.92,Z 524.691,A -85,B 0,C 180,E1 -7275.192,E2 -7275.192} C_VEL
LIN {X 0,Y 476.485,Z 538.185,A -85,B 0,C 180,E1 -7275.587,E2 -7275.587} C_VEL
LIN {X 0,Y 476.061,Z 550.545,A -85,B 0,C 180,E1 -7276.119,E2 -7276.119} C_VEL
LIN {X 0,Y 475.575,Z 563.273,A -85,B 0,C 180,E1 -7276.867,E2 -7276.867} C_VEL
LIN {X 0,Y 475.216,Z 574.177,A -85,B 0,C 180,E1 -7277.685,E2 -7277.685} C_VEL
LIN {X 0,Y 474.786,Z 583.887,A -85,B 0,C 180,E1 -7278.581,E2 -7278.581} C_VEL
LIN {X 0,Y 474.536,Z 592.53,A -85,B 0,C 180,E1 -7279.547,E2 -7279.547} C_VEL
LIN {X 0,Y 474.244,Z 601.886,A -85,B 0,C 180,E1 -7280.833,E2 -7280.833} C_VEL
LIN {X 0,Y 474.059,Z 609.415,A -85,B 0,C 180,E1 -7282.118,E2 -7282.118} C_VEL
LIN {X 0,Y 474.001,Z 615.53,A -85,B 0,C 180,E1 -7283.42,E2 -7283.42} C_VEL
LIN {X 0,Y 473.901,Z 620.838,A -85,B 0,C 180,E1 -7284.895,E2 -7284.895} C_VEL
LIN {X 0,Y 474,Z 623.232,A -85,B 0,C 180,E1 -7285.748,E2 -7285.748} C_VEL
LIN {X 0,Y 474.024,Z 625.167,A -85,B 0,C 180,E1 -7286.6,E2 -7286.6} C_VEL
LIN {X 0,Y 473.942,Z 626.613,A -85,B 0,C 180,E1 -7287.45,E2 -7287.45} C_VEL
LIN {X 0,Y 473.914,Z 627.621,A -85,B 0,C 180,E1 -7288.3,E2 -7288.3} C_VEL
LIN {X 0,Y 473.915,Z 628.221,A -85,B 0,C 180,E1 -7289.15,E2 -7289.15} C_VEL
LIN {X 0,Y 473.932,Z 628.411,A -85,B 0,C 180,E1 -7290,E2 -7290} C_VEL
LIN {X 0,Y 473.925,Z 628.138,A -85,B 0,C 180,E1 -7290.85,E2 -7290.85} C_VEL
LIN {X 0,Y 473.933,Z 627.447,A -85,B 0,C 180,E1 -7291.699,E2 -7291.699} C_VEL
LIN {X 0,Y 473.965,Z 626.344,A -85,B 0,C 180,E1 -7292.549,E2 -7292.549} C_VEL
LIN {X 0,Y 474.035,Z 623.849,A -85,B 0,C 180,E1 -7293.825,E2 -7293.825} C_VEL
LIN {X 0,Y 473.969,Z 620.283,A -85,B 0,C 180,E1 -7295.104,E2 -7295.104} C_VEL
LIN {X 0,Y 474.056,Z 615.703,A -85,B 0,C 180,E1 -7296.357,E2 -7296.357} C_VEL
LIN {X 0,Y 474.082,Z 609.625,A -85,B 0,C 180,E1 -7297.667,E2 -7297.667} C_VEL
LIN {X 0,Y 474.208,Z 602.165,A -85,B 0,C 180,E1 -7298.952,E2 -7298.952} C_VEL
LIN {X 0,Y 474.445,Z 592.863,A -85,B 0,C 180,E1 -7300.239,E2 -7300.239} C_VEL
LIN {X 0,Y 474.68,Z 583.33,A -85,B 0,C 180,E1 -7301.313,E2 -7301.313} C_VEL
LIN {X 0,Y 475.122,Z 573.645,A -85,B 0,C 180,E1 -7302.209,E2 -7302.209} C_VEL
LIN {X 0,Y 475.505,Z 562.796,A -85,B 0,C 180,E1 -7303.026,E2 -7303.026} C_VEL
LIN {X 0,Y 475.931,Z 550.185,A -85,B 0,C 180,E1 -7303.775,E2 -7303.775} C_VEL
LIN {X 0,Y 476.408,Z 536.957,A -85,B 0,C 180,E1 -7304.36,E2 -7304.36} C_VEL
LIN {X 0,Y 476.796,Z 523.769,A -85,B 0,C 180,E1 -7304.757,E2 -7304.757} C_VEL
LIN {X 0,Y 477.129,Z 494.735,A -85,B 0,C 180,E1 -7305.266,E2 -7305.266} C_VEL
LIN {X 0,Y 477.594,Z 433.824,A -85,B 0,C 180,E1 -7306.308,E2 -7306.308} C_VEL
LIN {X 0,Y 475.128,Z 410.026,A -85,B 0,C 180,E1 -7306.848,E2 -7306.848} C_VEL
LIN {X 0,Y 475.689,Z 389.232,A -85,B 0,C 180,E1 -7309.64,E2 -7309.64} C_VEL
LIN {X 0,Y 476.371,Z 369.562,A -85,B 0,C 180,E1 -7312.327,E2 -7312.327} C_VEL
LIN {X 0,Y 477.19,Z 348.48,A -85,B 0,C 180,E1 -7315.284,E2 -7315.284} C_VEL
LIN {X 0,Y 477.655,Z 337.243,A -85,B 0,C 180,E1 -7316.9,E2 -7316.9} C_VEL
LIN {X 0,Y 475.856,Z 327.651,A -85,B 0,C 180,E1 -7318.444,E2 -7318.444} C_VEL
LIN {X 0,Y 474.654,Z 322.363,A -85,B 0,C 180,E1 -7319.371,E2 -7319.371} C_VEL
LIN {X 0,Y 474.617,Z 322.37,A -85,B 0,C 180,E1 -7322.43,E2 -7322.43} C_VEL
LIN {X 0,Y 474.613,Z 322.365,A -85,B 0,C 180,E1 -7325.468,E2 -7325.468} C_VEL
LIN {X 0,Y 474.61,Z 322.369,A -85,B 0,C 180,E1 -7328.458,E2 -7328.458} C_VEL
LIN {X 0,Y 474.606,Z 322.368,A -85,B 0,C 180,E1 -7331.787,E2 -7331.787} C_VEL
LIN {X 0,Y 474.618,Z 322.364,A -85,B 0,C 180,E1 -7334.702,E2 -7334.702} C_VEL
LIN {X 0,Y 474.587,Z 322.37,A -85,B 0,C 180,E1 -7337.769,E2 -7337.769} C_VEL
LIN {X 0,Y 474.62,Z 322.364,A -85,B 0,C 180,E1 -7340.451,E2 -7340.451} C_VEL
LIN {X 0,Y 474.572,Z 322.37,A -85,B 0,C 180,E1 -7343.675,E2 -7343.675} C_VEL
LIN {X 0,Y 474.617,Z 322.361,A -85,B 0,C 180,E1 -7346.777,E2 -7346.777} C_VEL
LIN {X 0,Y 474.589,Z 322.371,A -85,B 0,C 180,E1 -7349.768,E2 -7349.768} C_VEL
LIN {X 0,Y 474.603,Z 322.364,A -85,B 0,C 180,E1 -7352.684,E2 -7352.684} C_VEL
LIN {X 0,Y 474.623,Z 322.368,A -85,B 0,C 180,E1 -7355.505,E2 -7355.505} C_VEL
LIN {X 0,Y 474.64,Z 322.364,A -85,B 0,C 180,E1 -7359.184,E2 -7359.184} C_VEL
LIN {X 0,Y 474.621,Z 322.367,A -85,B 0,C 180,E1 -7361.883,E2 -7361.883} C_VEL
LIN {X 0,Y 474.699,Z 322.356,A -85,B 0,C 180,E1 -7364.544,E2 -7364.544} C_VEL
LIN {X 0,Y 474.655,Z 322.365,A -85,B 0,C 180,E1 -7365.532,E2 -7365.532} C_VEL
LIN {X 0,Y 478.123,Z 332.101,A -85,B 0,C 180,E1 -7365.867,E2 -7365.867} C_VEL
LIN {X 0,Y 477.181,Z 414.011,A -85,B 0,C 180,E1 -7367.317,E2 -7367.317} C_VEL
LIN {X 0,Y 477.144,Z 426.874,A -85,B 0,C 180,E1 -7367.722,E2 -7367.722} C_VEL
LIN {X 0,Y 476.923,Z 438.786,A -85,B 0,C 180,E1 -7368.255,E2 -7368.255} C_VEL
LIN {X 0,Y 476.696,Z 450.32,A -85,B 0,C 180,E1 -7368.95,E2 -7368.95} C_VEL
LIN {X 0,Y 476.288,Z 461.459,A -85,B 0,C 180,E1 -7369.801,E2 -7369.801} C_VEL
LIN {X 0,Y 475.953,Z 471.484,A -85,B 0,C 180,E1 -7370.759,E2 -7370.759} C_VEL
LIN {X 0,Y 475.569,Z 480.009,A -85,B 0,C 180,E1 -7371.758,E2 -7371.758} C_VEL
LIN {X 0,Y 475.197,Z 488.692,A -85,B 0,C 180,E1 -7373.014,E2 -7373.014} C_VEL
LIN {X 0,Y 475.027,Z 495.647,A -85,B 0,C 180,E1 -7374.268,E2 -7374.268} C_VEL
LIN {X 0,Y 474.706,Z 500.446,A -85,B 0,C 180,E1 -7375.329,E2 -7375.329} C_VEL
LIN {X 0,Y 474.44,Z 505.069,A -85,B 0,C 180,E1 -7376.603,E2 -7376.603} C_VEL
LIN {X 0,Y 474.288,Z 507.544,A -85,B 0,C 180,E1 -7377.452,E2 -7377.452} C_VEL
LIN {X 0,Y 474.346,Z 509.484,A -85,B 0,C 180,E1 -7378.302,E2 -7378.302} C_VEL
LIN {X 0,Y 474.252,Z 511.032,A -85,B 0,C 180,E1 -7379.15,E2 -7379.15} C_VEL
LIN {X 0,Y 474.22,Z 512.171,A -85,B 0,C 180,E1 -7380,E2 -7380} C_VEL
LIN {X 0,Y 474.223,Z 512.864,A -85,B 0,C 180,E1 -7380.849,E2 -7380.849} C_VEL
LIN {X 0,Y 474.055,Z 513.173,A -85,B 0,C 180,E1 -7381.699,E2 -7381.699} C_VEL
LIN {X 0,Y 474.086,Z 513.068,A -85,B 0,C 180,E1 -7382.549,E2 -7382.549} C_VEL
LIN {X 0,Y 474.153,Z 512.568,A -85,B 0,C 180,E1 -7383.399,E2 -7383.399} C_VEL
LIN {X 0,Y 474.215,Z 511.627,A -85,B 0,C 180,E1 -7384.249,E2 -7384.249} C_VEL
LIN {X 0,Y 474.238,Z 510.288,A -85,B 0,C 180,E1 -7385.101,E2 -7385.101} C_VEL
LIN {X 0,Y 474.36,Z 507.472,A -85,B 0,C 180,E1 -7386.379,E2 -7386.379} C_VEL
LIN {X 0,Y 474.484,Z 503.62,A -85,B 0,C 180,E1 -7387.66,E2 -7387.66} C_VEL
LIN {X 0,Y 474.666,Z 498.612,A -85,B 0,C 180,E1 -7388.943,E2 -7388.943} C_VEL
LIN {X 0,Y 474.868,Z 492.301,A -85,B 0,C 180,E1 -7390.229,E2 -7390.229} C_VEL
LIN {X 0,Y 475.184,Z 484.382,A -85,B 0,C 180,E1 -7391.517,E2 -7391.517} C_VEL
LIN {X 0,Y 475.522,Z 475.175,A -85,B 0,C 180,E1 -7392.721,E2 -7392.721} C_VEL
LIN {X 0,Y 475.878,Z 465.234,A -85,B 0,C 180,E1 -7393.776,E2 -7393.776} C_VEL
LIN {X 0,Y 476.244,Z 455.168,A -85,B 0,C 180,E1 -7394.638,E2 -7394.638} C_VEL
LIN {X 0,Y 476.591,Z 444.205,A -85,B 0,C 180,E1 -7395.392,E2 -7395.392} C_VEL
LIN {X 0,Y 476.889,Z 432.118,A -85,B 0,C 180,E1 -7396.04,E2 -7396.04} C_VEL
LIN {X 0,Y 477.068,Z 419.323,A -85,B 0,C 180,E1 -7396.542,E2 -7396.542} C_VEL
LIN {X 0,Y 477.21,Z 406.471,A -85,B 0,C 180,E1 -7396.869,E2 -7396.869} C_VEL
LIN {X 0,Y 477.754,Z 331.673,A -85,B 0,C 180,E1 -7398.114,E2 -7398.114} C_VEL
LIN {X 0,Y 474.67,Z 322.361,A -85,B 0,C 180,E1 -7398.399,E2 -7398.399} C_VEL
LIN {X 0,Y 474.636,Z 322.361,A -85,B 0,C 180,E1 -7401.116,E2 -7401.116} C_VEL
LIN {X 0,Y 474.656,Z 322.361,A -85,B 0,C 180,E1 -7404.493,E2 -7404.493} C_VEL
LIN {X 0,Y 474.682,Z 322.354,A -85,B 0,C 180,E1 -7407.334,E2 -7407.334} C_VEL
LIN {X 0,Y 474.604,Z 322.365,A -85,B 0,C 180,E1 -7410.23,E2 -7410.23} C_VEL
LIN {X 0,Y 474.624,Z 322.361,A -85,B 0,C 180,E1 -7413.221,E2 -7413.221} C_VEL
LIN {X 0,Y 474.588,Z 322.368,A -85,B 0,C 180,E1 -7416.323,E2 -7416.323} C_VEL
LIN {X 0,Y 474.617,Z 322.361,A -85,B 0,C 180,E1 -7419.646,E2 -7419.646} C_VEL
LIN {X 0,Y 474.613,Z 322.364,A -85,B 0,C 180,E1 -7422.934,E2 -7422.934} C_VEL
LIN {X 0,Y 474.604,Z 322.365,A -85,B 0,C 180,E1 -7425.894,E2 -7425.894} C_VEL
LIN {X 0,Y 474.626,Z 322.361,A -85,B 0,C 180,E1 -7429.04,E2 -7429.04} C_VEL
LIN {X 0,Y 474.609,Z 322.363,A -85,B 0,C 180,E1 -7431.704,E2 -7431.704} C_VEL
LIN {X 0,Y 474.628,Z 322.363,A -85,B 0,C 180,E1 -7434.726,E2 -7434.726} C_VEL
LIN {X 0,Y 474.634,Z 322.361,A -85,B 0,C 180,E1 -7437.788,E2 -7437.788} C_VEL
LIN {X 0,Y 474.599,Z 322.365,A -85,B 0,C 180,E1 -7439.848,E2 -7439.848} C_VEL
LIN {X 0,Y 473.924,Z 322.452,A -85,B 0,C 180,E1 -7440.557,E2 -7440.557} C_VEL
LIN {X 0,Y 471.092,Z 322.802,A -85,B 0,C 180,E1 -7441.709,E2 -7441.709} C_VEL
LIN {X 0,Y 468.704,Z 323.102,A -85,B 0,C 180,E1 -7442.638,E2 -7442.638} C_VEL
LIN {X 0,Y 467.679,Z 323.226,A -85,B 0,C 180,E1 -7443.355,E2 -7443.355} C_VEL
LIN {X 0,Y 467.595,Z 323.236,A -85,B 0,C 180,E1 -7443.598,E2 -7443.598} C_VEL
LIN {X 0,Y 467.59,Z 323.242,A -85,B 0,C 180,E1 -7446.468,E2 -7446.468} C_VEL
LIN {X 0,Y 467.62,Z 323.235,A -85,B 0,C 180,E1 -7449.777,E2 -7449.777} C_VEL
LIN {X 0,Y 467.606,Z 323.239,A -85,B 0,C 180,E1 -7452.507,E2 -7452.507} C_VEL
LIN {X 0,Y 467.604,Z 323.235,A -85,B 0,C 180,E1 -7455.196,E2 -7455.196} C_VEL
LIN {X 0,Y 467.653,Z 323.232,A -85,B 0,C 180,E1 -7457.855,E2 -7457.855} C_VEL
LIN {X 0,Y 467.679,Z 323.226,A -85,B 0,C 180,E1 -7461.357,E2 -7461.357} C_VEL
LIN {X 0,Y 467.741,Z 323.222,A -85,B 0,C 180,E1 -7463.963,E2 -7463.963} C_VEL
LIN {X 0,Y 467.858,Z 323.205,A -85,B 0,C 180,E1 -7467.417,E2 -7467.417} C_VEL
LIN {X 0,Y 467.881,Z 323.206,A -85,B 0,C 180,E1 -7470,E2 -7470} C_VEL
LIN {X 0,Y 467.857,Z 323.205,A -85,B 0,C 180,E1 -7472.583,E2 -7472.583} C_VEL
LIN {X 0,Y 467.741,Z 323.224,A -85,B 0,C 180,E1 -7476.038,E2 -7476.038} C_VEL
LIN {X 0,Y 467.679,Z 323.227,A -85,B 0,C 180,E1 -7478.643,E2 -7478.643} C_VEL
LIN {X 0,Y 467.654,Z 323.234,A -85,B 0,C 180,E1 -7482.146,E2 -7482.146} C_VEL
LIN {X 0,Y 467.637,Z 323.234,A -85,B 0,C 180,E1 -7485.695,E2 -7485.695} C_VEL
LIN {X 0,Y 467.616,Z 323.234,A -85,B 0,C 180,E1 -7488.765,E2 -7488.765} C_VEL
LIN {X 0,Y 467.579,Z 323.24,A -85,B 0,C 180,E1 -7491.269,E2 -7491.269} C_VEL
LIN {X 0,Y 467.573,Z 323.245,A -85,B 0,C 180,E1 -7493.944,E2 -7493.944} C_VEL
LIN {X 0,Y 467.615,Z 323.234,A -85,B 0,C 180,E1 -7496.801,E2 -7496.801} C_VEL
LIN {X 0,Y 467.553,Z 323.246,A -85,B 0,C 180,E1 -7499.739,E2 -7499.739} C_VEL
LIN {X 0,Y 467.582,Z 323.238,A -85,B 0,C 180,E1 -7502.759,E2 -7502.759} C_VEL
LIN {X 0,Y 467.556,Z 323.247,A -85,B 0,C 180,E1 -7505.89,E2 -7505.89} C_VEL
LIN {X 0,Y 467.582,Z 323.24,A -85,B 0,C 180,E1 -7509.145,E2 -7509.145} C_VEL
LIN {X 0,Y 467.586,Z 323.238,A -85,B 0,C 180,E1 -7512.568,E2 -7512.568} C_VEL
LIN {X 0,Y 467.566,Z 323.242,A -85,B 0,C 180,E1 -7515.053,E2 -7515.053} C_VEL
LIN {X 0,Y 467.589,Z 323.241,A -85,B 0,C 180,E1 -7517.441,E2 -7517.441} C_VEL
LIN {X 0,Y 467.561,Z 323.242,A -85,B 0,C 180,E1 -7520.854,E2 -7520.854} C_VEL
LIN {X 0,Y 467.56,Z 323.242,A -85,B 0,C 180,E1 -7524.262,E2 -7524.262} C_VEL
LIN {X 0,Y 467.581,Z 323.242,A -85,B 0,C 180,E1 -7527.322,E2 -7527.322} C_VEL
LIN {X 0,Y 467.571,Z 323.24,A -85,B 0,C 180,E1 -7530.668,E2 -7530.668} C_VEL
LIN {X 0,Y 467.618,Z 323.238,A -85,B 0,C 180,E1 -7533.2,E2 -7533.2} C_VEL
LIN {X 0,Y 467.668,Z 323.412,A -85,B 0,C 180,E1 -7535.491,E2 -7535.491} C_VEL
LIN {X 0,Y 470.98,Z 333.354,A -85,B 0,C 180,E1 -7535.778,E2 -7535.778} C_VEL
LIN {X 0,Y 470.293,Z 411.573,A -85,B 0,C 180,E1 -7537.108,E2 -7537.108} C_VEL
LIN {X 0,Y 470.146,Z 423.059,A -85,B 0,C 180,E1 -7537.448,E2 -7537.448} C_VEL
LIN {X 0,Y 469.948,Z 435.898,A -85,B 0,C 180,E1 -7538.004,E2 -7538.004} C_VEL
LIN {X 0,Y 469.616,Z 448.214,A -85,B 0,C 180,E1 -7538.721,E2 -7538.721} C_VEL
LIN {X 0,Y 469.254,Z 458.784,A -85,B 0,C 180,E1 -7539.508,E2 -7539.508} C_VEL
LIN {X 0,Y 468.85,Z 469.578,A -85,B 0,C 180,E1 -7540.518,E2 -7540.518} C_VEL
LIN {X 0,Y 468.423,Z 479.278,A -85,B 0,C 180,E1 -7541.635,E2 -7541.635} C_VEL
LIN {X 0,Y 468.117,Z 487.167,A -85,B 0,C 180,E1 -7542.752,E2 -7542.752} C_VEL
LIN {X 0,Y 467.781,Z 494.661,A -85,B 0,C 180,E1 -7544.061,E2 -7544.061} C_VEL
LIN {X 0,Y 467.551,Z 499.953,A -85,B 0,C 180,E1 -7545.195,E2 -7545.195} C_VEL
LIN {X 0,Y 467.379,Z 504.904,A -85,B 0,C 180,E1 -7546.522,E2 -7546.522} C_VEL
LIN {X 0,Y 467.299,Z 508.667,A -85,B 0,C 180,E1 -7547.846,E2 -7547.846} C_VEL
LIN {X 0,Y 467.209,Z 510.603,A -85,B 0,C 180,E1 -7548.723,E2 -7548.723} C_VEL
LIN {X 0,Y 467.106,Z 512.049,A -85,B 0,C 180,E1 -7549.599,E2 -7549.599} C_VEL
LIN {X 0,Y 467.12,Z 513.076,A -85,B 0,C 180,E1 -7550.474,E2 -7550.474} C_VEL
LIN {X 0,Y 467.134,Z 513.71,A -85,B 0,C 180,E1 -7551.347,E2 -7551.347} C_VEL
LIN {X 0,Y 467.145,Z 513.89,A -85,B 0,C 180,E1 -7552.219,E2 -7552.219} C_VEL
LIN {X 0,Y 467.227,Z 513.65,A -85,B 0,C 180,E1 -7553.11,E2 -7553.11} C_VEL
LIN {X 0,Y 467.232,Z 513.053,A -85,B 0,C 180,E1 -7553.956,E2 -7553.956} C_VEL
LIN {X 0,Y 467.275,Z 512.01,A -85,B 0,C 180,E1 -7554.823,E2 -7554.823} C_VEL
LIN {X 0,Y 467.27,Z 510.546,A -85,B 0,C 180,E1 -7555.688,E2 -7555.688} C_VEL
LIN {X 0,Y 467.389,Z 507.535,A -85,B 0,C 180,E1 -7556.984,E2 -7556.984} C_VEL
LIN {X 0,Y 467.56,Z 503.464,A -85,B 0,C 180,E1 -7558.278,E2 -7558.278} C_VEL
LIN {X 0,Y 467.816,Z 498.211,A -85,B 0,C 180,E1 -7559.57,E2 -7559.57} C_VEL
LIN {X 0,Y 468.19,Z 491.606,A -85,B 0,C 180,E1 -7560.861,E2 -7560.861} C_VEL
LIN {X 0,Y 468.568,Z 483.323,A -85,B 0,C 180,E1 -7562.149,E2 -7562.149} C_VEL
LIN {X 0,Y 468.952,Z 474.838,A -85,B 0,C 180,E1 -7563.222,E2 -7563.222} C_VEL
LIN {X 0,Y 469.305,Z 465.551,A -85,B 0,C 180,E1 -7564.187,E2 -7564.187} C_VEL
LIN {X 0,Y 469.643,Z 455.362,A -85,B 0,C 180,E1 -7565.044,E2 -7565.044} C_VEL
LIN {X 0,Y 469.984,Z 444.165,A -85,B 0,C 180,E1 -7565.794,E2 -7565.794} C_VEL
LIN {X 0,Y 470.24,Z 431.679,A -85,B 0,C 180,E1 -7566.436,E2 -7566.436} C_VEL
LIN {X 0,Y 470.394,Z 419.102,A -85,B 0,C 180,E1 -7566.892,E2 -7566.892} C_VEL
LIN {X 0,Y 470.483,Z 406.314,A -85,B 0,C 180,E1 -7567.187,E2 -7567.187} C_VEL
LIN {X 0,Y 471.38,Z 333.514,A -85,B 0,C 180,E1 -7568.453,E2 -7568.453} C_VEL
LIN {X 0,Y 467.635,Z 323.24,A -85,B 0,C 180,E1 -7568.815,E2 -7568.815} C_VEL
LIN {X 0,Y 467.647,Z 323.237,A -85,B 0,C 180,E1 -7572.351,E2 -7572.351} C_VEL
LIN {X 0,Y 467.628,Z 323.236,A -85,B 0,C 180,E1 -7575.874,E2 -7575.874} C_VEL
LIN {X 0,Y 467.544,Z 323.247,A -85,B 0,C 180,E1 -7579.312,E2 -7579.312} C_VEL
LIN {X 0,Y 467.523,Z 323.253,A -85,B 0,C 180,E1 -7582.075,E2 -7582.075} C_VEL
LIN {X 0,Y 467.554,Z 323.244,A -85,B 0,C 180,E1 -7584.891,E2 -7584.891} C_VEL
LIN {X 0,Y 467.545,Z 323.246,A -85,B 0,C 180,E1 -7587.774,E2 -7587.774} C_VEL
LIN {X 0,Y 467.547,Z 323.243,A -85,B 0,C 180,E1 -7591.04,E2 -7591.04} C_VEL
LIN {X 0,Y 467.579,Z 323.242,A -85,B 0,C 180,E1 -7594.24,E2 -7594.24} C_VEL
LIN {X 0,Y 467.52,Z 323.244,A -85,B 0,C 180,E1 -7597.181,E2 -7597.181} C_VEL
LIN {X 0,Y 467.56,Z 323.242,A -85,B 0,C 180,E1 -7600.267,E2 -7600.267} C_VEL
LIN {X 0,Y 467.548,Z 323.247,A -85,B 0,C 180,E1 -7603.746,E2 -7603.746} C_VEL
LIN {X 0,Y 467.55,Z 323.245,A -85,B 0,C 180,E1 -7606.254,E2 -7606.254} C_VEL
LIN {X 0,Y 467.563,Z 323.246,A -85,B 0,C 180,E1 -7609.733,E2 -7609.733} C_VEL
LIN {X 0,Y 467.545,Z 323.243,A -85,B 0,C 180,E1 -7612.815,E2 -7612.815} C_VEL
LIN {X 0,Y 467.58,Z 323.244,A -85,B 0,C 180,E1 -7615.76,E2 -7615.76} C_VEL
LIN {X 0,Y 467.572,Z 323.242,A -85,B 0,C 180,E1 -7618.955,E2 -7618.955} C_VEL
LIN {X 0,Y 467.659,Z 323.418,A -85,B 0,C 180,E1 -7620.207,E2 -7620.207} C_VEL
LIN {X 0,Y 471.094,Z 339.293,A -85,B 0,C 180,E1 -7622.694,E2 -7622.694} C_VEL
LIN {X 0,Y 471.055,Z 345.848,A -85,B 0,C 180,E1 -7623.637,E2 -7623.637} C_VEL
LIN {X 0,Y 469.977,Z 368.99,A -85,B 0,C 180,E1 -7626.887,E2 -7626.887} C_VEL
LIN {X 0,Y 469.125,Z 390.314,A -85,B 0,C 180,E1 -7629.844,E2 -7629.844} C_VEL
LIN {X 0,Y 468.403,Z 411.554,A -85,B 0,C 180,E1 -7632.763,E2 -7632.763} C_VEL
LIN {X 0,Y 468.353,Z 413.362,A -85,B 0,C 180,E1 -7633.01,E2 -7633.01} C_VEL
LIN {X 0,Y 470.925,Z 436.072,A -85,B 0,C 180,E1 -7633.497,E2 -7633.497} C_VEL
LIN {X 0,Y 470.008,Z 523.776,A -85,B 0,C 180,E1 -7634.997,E2 -7634.997} C_VEL
LIN {X 0,Y 469.546,Z 537.287,A -85,B 0,C 180,E1 -7635.397,E2 -7635.397} C_VEL
LIN {X 0,Y 469.082,Z 550.196,A -85,B 0,C 180,E1 -7635.964,E2 -7635.964} C_VEL
LIN {X 0,Y 468.546,Z 562.019,A -85,B 0,C 180,E1 -7636.666,E2 -7636.666} C_VEL
LIN {X 0,Y 468.176,Z 573.247,A -85,B 0,C 180,E1 -7637.517,E2 -7637.517} C_VEL
LIN {X 0,Y 467.766,Z 582.802,A -85,B 0,C 180,E1 -7638.407,E2 -7638.407} C_VEL
LIN {X 0,Y 467.511,Z 591.506,A -85,B 0,C 180,E1 -7639.388,E2 -7639.388} C_VEL
LIN {X 0,Y 467.193,Z 599.518,A -85,B 0,C 180,E1 -7640.475,E2 -7640.475} C_VEL
LIN {X 0,Y 467.002,Z 607.339,A -85,B 0,C 180,E1 -7641.78,E2 -7641.78} C_VEL
LIN {X 0,Y 466.915,Z 613.619,A -85,B 0,C 180,E1 -7643.084,E2 -7643.084} C_VEL
LIN {X 0,Y 466.894,Z 618.579,A -85,B 0,C 180,E1 -7644.385,E2 -7644.385} C_VEL
LIN {X 0,Y 466.94,Z 622.367,A -85,B 0,C 180,E1 -7645.684,E2 -7645.684} C_VEL
LIN {X 0,Y 466.976,Z 624.31,A -85,B 0,C 180,E1 -7646.549,E2 -7646.549} C_VEL
LIN {X 0,Y 466.887,Z 625.762,A -85,B 0,C 180,E1 -7647.412,E2 -7647.412} C_VEL
LIN {X 0,Y 466.861,Z 626.771,A -85,B 0,C 180,E1 -7648.275,E2 -7648.275} C_VEL
LIN {X 0,Y 466.864,Z 627.369,A -85,B 0,C 180,E1 -7649.137,E2 -7649.137} C_VEL
LIN {X 0,Y 466.884,Z 627.557,A -85,B 0,C 180,E1 -7650,E2 -7650} C_VEL
LIN {X 0,Y 466.875,Z 627.279,A -85,B 0,C 180,E1 -7650.862,E2 -7650.862} C_VEL
LIN {X 0,Y 466.881,Z 626.578,A -85,B 0,C 180,E1 -7651.725,E2 -7651.725} C_VEL
LIN {X 0,Y 466.911,Z 625.467,A -85,B 0,C 180,E1 -7652.588,E2 -7652.588} C_VEL
LIN {X 0,Y 466.992,Z 622.956,A -85,B 0,C 180,E1 -7653.883,E2 -7653.883} C_VEL
LIN {X 0,Y 466.9,Z 619.366,A -85,B 0,C 180,E1 -7655.182,E2 -7655.182} C_VEL
LIN {X 0,Y 466.982,Z 614.011,A -85,B 0,C 180,E1 -7656.639,E2 -7656.639} C_VEL
LIN {X 0,Y 467.042,Z 607.51,A -85,B 0,C 180,E1 -7658.001,E2 -7658.001} C_VEL
LIN {X 0,Y 467.182,Z 599.721,A -85,B 0,C 180,E1 -7659.306,E2 -7659.306} C_VEL
LIN {X 0,Y 467.471,Z 590.088,A -85,B 0,C 180,E1 -7660.613,E2 -7660.613} C_VEL
LIN {X 0,Y 467.829,Z 580.093,A -85,B 0,C 180,E1 -7661.701,E2 -7661.701} C_VEL
LIN {X 0,Y 468.208,Z 568.513,A -85,B 0,C 180,E1 -7662.723,E2 -7662.723} C_VEL
LIN {X 0,Y 468.669,Z 556.647,A -85,B 0,C 180,E1 -7663.551,E2 -7663.551} C_VEL
LIN {X 0,Y 469.259,Z 543.534,A -85,B 0,C 180,E1 -7664.252,E2 -7664.252} C_VEL
LIN {X 0,Y 469.681,Z 530.352,A -85,B 0,C 180,E1 -7664.764,E2 -7664.764} C_VEL
LIN {X 0,Y 470.042,Z 516.286,A -85,B 0,C 180,E1 -7665.113,E2 -7665.113} C_VEL
LIN {X 0,Y 470.874,Z 435.203,A -85,B 0,C 180,E1 -7666.525,E2 -7666.525} C_VEL
LIN {X 0,Y 468.164,Z 408.943,A -85,B 0,C 180,E1 -7667.135,E2 -7667.135} C_VEL
LIN {X 0,Y 468.699,Z 388.431,A -85,B 0,C 180,E1 -7669.946,E2 -7669.946} C_VEL
LIN {X 0,Y 469.452,Z 368.875,A -85,B 0,C 180,E1 -7672.674,E2 -7672.674} C_VEL
LIN {X 0,Y 470.321,Z 349.557,A -85,B 0,C 180,E1 -7675.443,E2 -7675.443} C_VEL
LIN {X 0,Y 470.785,Z 338.443,A -85,B 0,C 180,E1 -7677.085,E2 -7677.085} C_VEL
LIN {X 0,Y 468.639,Z 327.727,A -85,B 0,C 180,E1 -7678.87,E2 -7678.87} C_VEL
LIN {X 0,Y 467.624,Z 323.239,A -85,B 0,C 180,E1 -7679.675,E2 -7679.675} C_VEL
LIN {X 0,Y 467.582,Z 323.246,A -85,B 0,C 180,E1 -7682.759,E2 -7682.759} C_VEL
LIN {X 0,Y 467.553,Z 323.246,A -85,B 0,C 180,E1 -7685.89,E2 -7685.89} C_VEL
LIN {X 0,Y 467.554,Z 323.244,A -85,B 0,C 180,E1 -7689.148,E2 -7689.148} C_VEL
LIN {X 0,Y 467.567,Z 323.243,A -85,B 0,C 180,E1 -7691.404,E2 -7691.404} C_VEL
LIN {X 0,Y 467.568,Z 323.241,A -85,B 0,C 180,E1 -7695.052,E2 -7695.052} C_VEL
LIN {X 0,Y 467.564,Z 323.242,A -85,B 0,C 180,E1 -7698.725,E2 -7698.725} C_VEL
LIN {X 0,Y 467.543,Z 323.247,A -85,B 0,C 180,E1 -7701.953,E2 -7701.953} C_VEL
LIN {X 0,Y 467.552,Z 323.242,A -85,B 0,C 180,E1 -7705.166,E2 -7705.166} C_VEL
LIN {X 0,Y 467.559,Z 323.245,A -85,B 0,C 180,E1 -7708.258,E2 -7708.258} C_VEL
LIN {X 0,Y 467.541,Z 323.246,A -85,B 0,C 180,E1 -7711.248,E2 -7711.248} C_VEL
LIN {X 0,Y 467.563,Z 323.243,A -85,B 0,C 180,E1 -7714.405,E2 -7714.405} C_VEL
LIN {X 0,Y 467.553,Z 323.245,A -85,B 0,C 180,E1 -7716.994,E2 -7716.994} C_VEL
LIN {X 0,Y 467.589,Z 323.242,A -85,B 0,C 180,E1 -7719.775,E2 -7719.775} C_VEL
LIN {X 0,Y 467.578,Z 323.241,A -85,B 0,C 180,E1 -7722.505,E2 -7722.505} C_VEL
LIN {X 0,Y 467.616,Z 323.243,A -85,B 0,C 180,E1 -7725.235,E2 -7725.235} C_VEL
LIN {X 0,Y 471.438,Z 333.757,A -85,B 0,C 180,E1 -7725.616,E2 -7725.616} C_VEL
LIN {X 0,Y 470.371,Z 414.23,A -85,B 0,C 180,E1 -7727.076,E2 -7727.076} C_VEL
LIN {X 0,Y 470.342,Z 427.993,A -85,B 0,C 180,E1 -7727.514,E2 -7727.514} C_VEL
LIN {X 0,Y 470.098,Z 439.327,A -85,B 0,C 180,E1 -7728.028,E2 -7728.028} C_VEL
LIN {X 0,Y 469.883,Z 450.179,A -85,B 0,C 180,E1 -7728.678,E2 -7728.678} C_VEL
LIN {X 0,Y 469.471,Z 461.499,A -85,B 0,C 180,E1 -7729.542,E2 -7729.542} C_VEL
LIN {X 0,Y 469.111,Z 471.695,A -85,B 0,C 180,E1 -7730.514,E2 -7730.514} C_VEL
LIN {X 0,Y 468.645,Z 481.03,A -85,B 0,C 180,E1 -7731.614,E2 -7731.614} C_VEL
LIN {X 0,Y 468.257,Z 489.773,A -85,B 0,C 180,E1 -7732.901,E2 -7732.901} C_VEL
LIN {X 0,Y 468.044,Z 496.743,A -85,B 0,C 180,E1 -7734.182,E2 -7734.182} C_VEL
LIN {X 0,Y 467.731,Z 501.503,A -85,B 0,C 180,E1 -7735.259,E2 -7735.259} C_VEL
LIN {X 0,Y 467.428,Z 506.097,A -85,B 0,C 180,E1 -7736.552,E2 -7736.552} C_VEL
LIN {X 0,Y 467.267,Z 508.546,A -85,B 0,C 180,E1 -7737.413,E2 -7737.413} C_VEL
LIN {X 0,Y 467.321,Z 510.468,A -85,B 0,C 180,E1 -7738.276,E2 -7738.276} C_VEL
LIN {X 0,Y 467.227,Z 511.996,A -85,B 0,C 180,E1 -7739.138,E2 -7739.138} C_VEL
LIN {X 0,Y 467.193,Z 513.11,A -85,B 0,C 180,E1 -7740,E2 -7740} C_VEL
LIN {X 0,Y 467.193,Z 513.77,A -85,B 0,C 180,E1 -7740.862,E2 -7740.862} C_VEL
LIN {X 0,Y 467.011,Z 514.058,A -85,B 0,C 180,E1 -7741.724,E2 -7741.724} C_VEL
LIN {X 0,Y 467.042,Z 513.929,A -85,B 0,C 180,E1 -7742.587,E2 -7742.587} C_VEL
LIN {X 0,Y 467.108,Z 513.392,A -85,B 0,C 180,E1 -7743.45,E2 -7743.45} C_VEL
LIN {X 0,Y 467.185,Z 512.414,A -85,B 0,C 180,E1 -7744.313,E2 -7744.313} C_VEL
LIN {X 0,Y 467.213,Z 511.046,A -85,B 0,C 180,E1 -7745.178,E2 -7745.178} C_VEL
LIN {X 0,Y 467.361,Z 509.257,A -85,B 0,C 180,E1 -7746.042,E2 -7746.042} C_VEL
LIN {X 0,Y 467.448,Z 505.835,A -85,B 0,C 180,E1 -7747.298,E2 -7747.298} C_VEL
LIN {X 0,Y 467.591,Z 501.031,A -85,B 0,C 180,E1 -7748.644,E2 -7748.644} C_VEL
LIN {X 0,Y 467.83,Z 493.93,A -85,B 0,C 180,E1 -7750.166,E2 -7750.166} C_VEL
LIN {X 0,Y 468.176,Z 486.224,A -85,B 0,C 180,E1 -7751.472,E2 -7751.472} C_VEL
LIN {X 0,Y 468.495,Z 477.773,A -85,B 0,C 180,E1 -7752.629,E2 -7752.629} C_VEL
LIN {X 0,Y 468.86,Z 467.526,A -85,B 0,C 180,E1 -7753.766,E2 -7753.766} C_VEL
LIN {X 0,Y 469.28,Z 456.48,A -85,B 0,C 180,E1 -7754.749,E2 -7754.749} C_VEL
LIN {X 0,Y 469.667,Z 445.63,A -85,B 0,C 180,E1 -7755.514,E2 -7755.514} C_VEL
LIN {X 0,Y 469.999,Z 432.583,A -85,B 0,C 180,E1 -7756.226,E2 -7756.226} C_VEL
LIN {X 0,Y 470.18,Z 419.547,A -85,B 0,C 180,E1 -7756.738,E2 -7756.738} C_VEL
LIN {X 0,Y 470.305,Z 406.811,A -85,B 0,C 180,E1 -7757.063,E2 -7757.063} C_VEL
LIN {X 0,Y 470.909,Z 333.128,A -85,B 0,C 180,E1 -7758.316,E2 -7758.316} C_VEL
LIN {X 0,Y 467.618,Z 323.24,A -85,B 0,C 180,E1 -7758.625,E2 -7758.625} C_VEL
LIN {X 0,Y 467.582,Z 323.239,A -85,B 0,C 180,E1 -7761.268,E2 -7761.268} C_VEL
LIN {X 0,Y 467.572,Z 323.239,A -85,B 0,C 180,E1 -7763.943,E2 -7763.943} C_VEL
LIN {X 0,Y 467.616,Z 323.239,A -85,B 0,C 180,E1 -7766.8,E2 -7766.8} C_VEL
LIN {X 0,Y 467.553,Z 323.241,A -85,B 0,C 180,E1 -7769.738,E2 -7769.738} C_VEL
LIN {X 0,Y 467.579,Z 323.244,A -85,B 0,C 180,E1 -7772.758,E2 -7772.758} C_VEL
LIN {X 0,Y 467.552,Z 323.242,A -85,B 0,C 180,E1 -7775.889,E2 -7775.889} C_VEL
LIN {X 0,Y 467.559,Z 323.242,A -85,B 0,C 180,E1 -7779.146,E2 -7779.146} C_VEL
LIN {X 0,Y 467.585,Z 323.244,A -85,B 0,C 180,E1 -7782.567,E2 -7782.567} C_VEL
LIN {X 0,Y 467.564,Z 323.241,A -85,B 0,C 180,E1 -7785.052,E2 -7785.052} C_VEL
LIN {X 0,Y 467.587,Z 323.237,A -85,B 0,C 180,E1 -7787.44,E2 -7787.44} C_VEL
LIN {X 0,Y 467.581,Z 323.24,A -85,B 0,C 180,E1 -7790.855,E2 -7790.855} C_VEL
LIN {X 0,Y 467.561,Z 323.245,A -85,B 0,C 180,E1 -7794.26,E2 -7794.26} C_VEL
LIN {X 0,Y 467.58,Z 323.238,A -85,B 0,C 180,E1 -7797.321,E2 -7797.321} C_VEL
LIN {X 0,Y 467.568,Z 323.243,A -85,B 0,C 180,E1 -7800.667,E2 -7800.667} C_VEL
LIN {X 0,Y 467.614,Z 323.234,A -85,B 0,C 180,E1 -7803.2,E2 -7803.2} C_VEL
LIN {X 0,Y 467.595,Z 323.236,A -85,B 0,C 180,E1 -7803.598,E2 -7803.598} C_VEL
LIN {X 0,Y 466.921,Z 323.326,A -85,B 0,C 180,E1 -7804.317,E2 -7804.317} C_VEL
LIN {X 0,Y 464.046,Z 323.679,A -85,B 0,C 180,E1 -7805.485,E2 -7805.485} C_VEL
LIN {X 0,Y 461.62,Z 323.986,A -85,B 0,C 180,E1 -7806.426,E2 -7806.426} C_VEL
LIN {X 0,Y 460.586,Z 324.11,A -85,B 0,C 180,E1 -7807.154,E2 -7807.154} C_VEL
LIN {X 0,Y 460.506,Z 324.12,A -85,B 0,C 180,E1 -7807.4,E2 -7807.4} C_VEL
LIN {X 0,Y 460.566,Z 324.118,A -85,B 0,C 180,E1 -7810.384,E2 -7810.384} C_VEL
LIN {X 0,Y 460.563,Z 324.112,A -85,B 0,C 180,E1 -7813.146,E2 -7813.146} C_VEL
LIN {X 0,Y 460.552,Z 324.116,A -85,B 0,C 180,E1 -7815.868,E2 -7815.868} C_VEL
LIN {X 0,Y 460.609,Z 324.109,A -85,B 0,C 180,E1 -7818.559,E2 -7818.559} C_VEL
LIN {X 0,Y 460.692,Z 324.101,A -85,B 0,C 180,E1 -7822.109,E2 -7822.109} C_VEL
LIN {X 0,Y 460.695,Z 324.097,A -85,B 0,C 180,E1 -7824.748,E2 -7824.748} C_VEL
LIN {X 0,Y 460.822,Z 324.081,A -85,B 0,C 180,E1 -7827.378,E2 -7827.378} C_VEL
LIN {X 0,Y 460.851,Z 324.081,A -85,B 0,C 180,E1 -7830,E2 -7830} C_VEL
LIN {X 0,Y 460.822,Z 324.081,A -85,B 0,C 180,E1 -7832.623,E2 -7832.623} C_VEL
LIN {X 0,Y 460.707,Z 324.1,A -85,B 0,C 180,E1 -7836.13,E2 -7836.13} C_VEL
LIN {X 0,Y 460.626,Z 324.105,A -85,B 0,C 180,E1 -7838.776,E2 -7838.776} C_VEL
LIN {X 0,Y 460.611,Z 324.108,A -85,B 0,C 180,E1 -7842.445,E2 -7842.445} C_VEL
LIN {X 0,Y 460.598,Z 324.114,A -85,B 0,C 180,E1 -7845.998,E2 -7845.998} C_VEL
LIN {X 0,Y 460.569,Z 324.112,A -85,B 0,C 180,E1 -7848.902,E2 -7848.902} C_VEL
LIN {X 0,Y 460.514,Z 324.121,A -85,B 0,C 180,E1 -7851.486,E2 -7851.486} C_VEL
LIN {X 0,Y 460.542,Z 324.117,A -85,B 0,C 180,E1 -7854.333,E2 -7854.333} C_VEL
LIN {X 0,Y 460.578,Z 324.112,A -85,B 0,C 180,E1 -7857.244,E2 -7857.244} C_VEL
LIN {X 0,Y 460.51,Z 324.121,A -85,B 0,C 180,E1 -7860.24,E2 -7860.24} C_VEL
LIN {X 0,Y 460.529,Z 324.119,A -85,B 0,C 180,E1 -7863.325,E2 -7863.325} C_VEL
LIN {X 0,Y 460.478,Z 324.123,A -85,B 0,C 180,E1 -7866.53,E2 -7866.53} C_VEL
LIN {X 0,Y 460.558,Z 324.119,A -85,B 0,C 180,E1 -7869.86,E2 -7869.86} C_VEL
LIN {X 0,Y 460.512,Z 324.12,A -85,B 0,C 180,E1 -7872.901,E2 -7872.901} C_VEL
LIN {X 0,Y 460.509,Z 324.124,A -85,B 0,C 180,E1 -7875.831,E2 -7875.831} C_VEL
LIN {X 0,Y 460.531,Z 324.118,A -85,B 0,C 180,E1 -7878.989,E2 -7878.989} C_VEL
LIN {X 0,Y 460.519,Z 324.12,A -85,B 0,C 180,E1 -7881.267,E2 -7881.267} C_VEL
LIN {X 0,Y 460.509,Z 324.12,A -85,B 0,C 180,E1 -7884.555,E2 -7884.555} C_VEL
LIN {X 0,Y 460.531,Z 324.122,A -85,B 0,C 180,E1 -7887.716,E2 -7887.716} C_VEL
LIN {X 0,Y 460.541,Z 324.117,A -85,B 0,C 180,E1 -7890.77,E2 -7890.77} C_VEL
LIN {X 0,Y 460.562,Z 324.116,A -85,B 0,C 180,E1 -7893.735,E2 -7893.735} C_VEL
LIN {X 0,Y 460.585,Z 324.114,A -85,B 0,C 180,E1 -7895.238,E2 -7895.238} C_VEL
LIN {X 0,Y 464.233,Z 335.519,A -85,B 0,C 180,E1 -7895.589,E2 -7895.589} C_VEL
LIN {X 0,Y 463.379,Z 411.181,A -85,B 0,C 180,E1 -7896.894,E2 -7896.894} C_VEL
LIN {X 0,Y 463.255,Z 423.898,A -85,B 0,C 180,E1 -7897.271,E2 -7897.271} C_VEL
LIN {X 0,Y 463.055,Z 435.951,A -85,B 0,C 180,E1 -7897.794,E2 -7897.794} C_VEL
LIN {X 0,Y 462.72,Z 448.354,A -85,B 0,C 180,E1 -7898.519,E2 -7898.519} C_VEL
LIN {X 0,Y 462.325,Z 458.899,A -85,B 0,C 180,E1 -7899.303,E2 -7899.303} C_VEL
LIN {X 0,Y 461.921,Z 469.858,A -85,B 0,C 180,E1 -7900.329,E2 -7900.329} C_VEL
LIN {X 0,Y 461.521,Z 478.752,A -85,B 0,C 180,E1 -7901.351,E2 -7901.351} C_VEL
LIN {X 0,Y 461.155,Z 486.902,A -85,B 0,C 180,E1 -7902.483,E2 -7902.483} C_VEL
LIN {X 0,Y 460.853,Z 493.855,A -85,B 0,C 180,E1 -7903.659,E2 -7903.659} C_VEL
LIN {X 0,Y 460.568,Z 500.117,A -85,B 0,C 180,E1 -7904.965,E2 -7904.965} C_VEL
LIN {X 0,Y 460.376,Z 505.22,A -85,B 0,C 180,E1 -7906.313,E2 -7906.313} C_VEL
LIN {X 0,Y 460.271,Z 509.358,A -85,B 0,C 180,E1 -7907.753,E2 -7907.753} C_VEL
LIN {X 0,Y 460.19,Z 511.134,A -85,B 0,C 180,E1 -7908.549,E2 -7908.549} C_VEL
LIN {X 0,Y 460.072,Z 512.697,A -85,B 0,C 180,E1 -7909.438,E2 -7909.438} C_VEL
LIN {X 0,Y 460.098,Z 514.479,A -85,B 0,C 180,E1 -7911.214,E2 -7911.214} C_VEL
LIN {X 0,Y 460.115,Z 514.766,A -85,B 0,C 180,E1 -7912.099,E2 -7912.099} C_VEL
LIN {X 0,Y 460.183,Z 514.552,A -85,B 0,C 180,E1 -7913.073,E2 -7913.073} C_VEL
LIN {X 0,Y 460.247,Z 513.088,A -85,B 0,C 180,E1 -7914.744,E2 -7914.744} C_VEL
LIN {X 0,Y 460.238,Z 511.686,A -85,B 0,C 180,E1 -7915.622,E2 -7915.622} C_VEL
LIN {X 0,Y 460.362,Z 508.778,A -85,B 0,C 180,E1 -7916.938,E2 -7916.938} C_VEL
LIN {X 0,Y 460.549,Z 504.809,A -85,B 0,C 180,E1 -7918.251,E2 -7918.251} C_VEL
LIN {X 0,Y 460.837,Z 499.66,A -85,B 0,C 180,E1 -7919.564,E2 -7919.564} C_VEL
LIN {X 0,Y 461.203,Z 493.183,A -85,B 0,C 180,E1 -7920.874,E2 -7920.874} C_VEL
LIN {X 0,Y 461.614,Z 485.103,A -85,B 0,C 180,E1 -7922.182,E2 -7922.182} C_VEL
LIN {X 0,Y 462.005,Z 476.814,A -85,B 0,C 180,E1 -7923.271,E2 -7923.271} C_VEL
LIN {X 0,Y 462.44,Z 466.657,A -85,B 0,C 180,E1 -7924.358,E2 -7924.358} C_VEL
LIN {X 0,Y 462.8,Z 456.553,A -85,B 0,C 180,E1 -7925.228,E2 -7925.228} C_VEL
LIN {X 0,Y 463.176,Z 445.417,A -85,B 0,C 180,E1 -7925.988,E2 -7925.988} C_VEL
LIN {X 0,Y 463.453,Z 433.028,A -85,B 0,C 180,E1 -7926.64,E2 -7926.64} C_VEL
LIN {X 0,Y 463.58,Z 420.708,A -85,B 0,C 180,E1 -7927.103,E2 -7927.103} C_VEL
LIN {X 0,Y 463.693,Z 406.84,A -85,B 0,C 180,E1 -7927.43,E2 -7927.43} C_VEL
LIN {X 0,Y 464.646,Z 335.05,A -85,B 0,C 180,E1 -7928.71,E2 -7928.71} C_VEL
LIN {X 0,Y 460.678,Z 324.695,A -85,B 0,C 180,E1 -7929.094,E2 -7929.094} C_VEL
LIN {X 0,Y 460.565,Z 324.119,A -85,B 0,C 180,E1 -7929.121,E2 -7929.121} C_VEL
LIN {X 0,Y 460.602,Z 324.114,A -85,B 0,C 180,E1 -7932.435,E2 -7932.435} C_VEL
LIN {X 0,Y 460.584,Z 324.114,A -85,B 0,C 180,E1 -7935.988,E2 -7935.988} C_VEL
LIN {X 0,Y 460.531,Z 324.123,A -85,B 0,C 180,E1 -7938.885,E2 -7938.885} C_VEL
LIN {X 0,Y 460.497,Z 324.126,A -85,B 0,C 180,E1 -7942.43,E2 -7942.43} C_VEL
LIN {X 0,Y 460.526,Z 324.121,A -85,B 0,C 180,E1 -7945.79,E2 -7945.79} C_VEL
LIN {X 0,Y 460.52,Z 324.118,A -85,B 0,C 180,E1 -7949.233,E2 -7949.233} C_VEL
LIN {X 0,Y 460.521,Z 324.123,A -85,B 0,C 180,E1 -7952.286,E2 -7952.286} C_VEL
LIN {X 0,Y 460.504,Z 324.118,A -85,B 0,C 180,E1 -7955.447,E2 -7955.447} C_VEL
LIN {X 0,Y 460.496,Z 324.119,A -85,B 0,C 180,E1 -7958.889,E2 -7958.889} C_VEL
LIN {X 0,Y 460.506,Z 324.12,A -85,B 0,C 180,E1 -7961.598,E2 -7961.598} C_VEL
LIN {X 0,Y 460.515,Z 324.119,A -85,B 0,C 180,E1 -7964.589,E2 -7964.589} C_VEL
LIN {X 0,Y 460.495,Z 324.127,A -85,B 0,C 180,E1 -7967.815,E2 -7967.815} C_VEL
LIN {X 0,Y 460.517,Z 324.122,A -85,B 0,C 180,E1 -7970.136,E2 -7970.136} C_VEL
LIN {X 0,Y 460.475,Z 324.128,A -85,B 0,C 180,E1 -7973.47,E2 -7973.47} C_VEL
LIN {X 0,Y 460.523,Z 324.119,A -85,B 0,C 180,E1 -7976.674,E2 -7976.674} C_VEL
LIN {X 0,Y 460.568,Z 324.179,A -85,B 0,C 180,E1 -7979.955,E2 -7979.955} C_VEL
LIN {X 0,Y 464.052,Z 340.077,A -85,B 0,C 180,E1 -7982.489,E2 -7982.489} C_VEL
LIN {X 0,Y 464.314,Z 343.434,A -85,B 0,C 180,E1 -7982.993,E2 -7982.993} C_VEL
LIN {X 0,Y 463.153,Z 366.511,A -85,B 0,C 180,E1 -7986.289,E2 -7986.289} C_VEL
LIN {X 0,Y 462.306,Z 386.195,A -85,B 0,C 180,E1 -7989.068,E2 -7989.068} C_VEL
LIN {X 0,Y 461.579,Z 405.824,A -85,B 0,C 180,E1 -7991.812,E2 -7991.812} C_VEL
LIN {X 0,Y 461.347,Z 412.686,A -85,B 0,C 180,E1 -7992.765,E2 -7992.765} C_VEL
LIN {X 0,Y 464.043,Z 437.691,A -85,B 0,C 180,E1 -7993.307,E2 -7993.307} C_VEL
LIN {X 0,Y 463.067,Z 523.863,A -85,B 0,C 180,E1 -7994.823,E2 -7994.823} C_VEL
LIN {X 0,Y 462.568,Z 537.813,A -85,B 0,C 180,E1 -7995.256,E2 -7995.256} C_VEL
LIN {X 0,Y 462.116,Z 549.79,A -85,B 0,C 180,E1 -7995.804,E2 -7995.804} C_VEL
LIN {X 0,Y 461.504,Z 562.325,A -85,B 0,C 180,E1 -7996.571,E2 -7996.571} C_VEL
LIN {X 0,Y 461.112,Z 573.293,A -85,B 0,C 180,E1 -7997.429,E2 -7997.429} C_VEL
LIN {X 0,Y 460.698,Z 582.752,A -85,B 0,C 180,E1 -7998.338,E2 -7998.338} C_VEL
LIN {X 0,Y 460.399,Z 592.159,A -85,B 0,C 180,E1 -7999.445,E2 -7999.445} C_VEL
LIN {X 0,Y 460.079,Z 601.303,A -85,B 0,C 180,E1 -8000.77,E2 -8000.77} C_VEL
LIN {X 0,Y 459.897,Z 608.656,A -85,B 0,C 180,E1 -8002.095,E2 -8002.095} C_VEL
LIN {X 0,Y 459.833,Z 614.583,A -85,B 0,C 180,E1 -8003.44,E2 -8003.44} C_VEL
LIN {X 0,Y 459.773,Z 619.068,A -85,B 0,C 180,E1 -8004.738,E2 -8004.738} C_VEL
LIN {X 0,Y 459.88,Z 621.481,A -85,B 0,C 180,E1 -8005.618,E2 -8005.618} C_VEL
LIN {X 0,Y 459.928,Z 623.433,A -85,B 0,C 180,E1 -8006.496,E2 -8006.496} C_VEL
LIN {X 0,Y 459.833,Z 624.897,A -85,B 0,C 180,E1 -8007.372,E2 -8007.372} C_VEL
LIN {X 0,Y 459.808,Z 625.909,A -85,B 0,C 180,E1 -8008.248,E2 -8008.248} C_VEL
LIN {X 0,Y 459.815,Z 626.509,A -85,B 0,C 180,E1 -8009.124,E2 -8009.124} C_VEL
LIN {X 0,Y 459.837,Z 626.696,A -85,B 0,C 180,E1 -8010,E2 -8010} C_VEL
LIN {X 0,Y 459.825,Z 626.419,A -85,B 0,C 180,E1 -8010.876,E2 -8010.876} C_VEL
LIN {X 0,Y 459.829,Z 625.712,A -85,B 0,C 180,E1 -8011.752,E2 -8011.752} C_VEL
LIN {X 0,Y 459.857,Z 624.591,A -85,B 0,C 180,E1 -8012.628,E2 -8012.628} C_VEL
LIN {X 0,Y 459.948,Z 622.065,A -85,B 0,C 180,E1 -8013.943,E2 -8013.943} C_VEL
LIN {X 0,Y 459.833,Z 618.455,A -85,B 0,C 180,E1 -8015.261,E2 -8015.261} C_VEL
LIN {X 0,Y 459.908,Z 613.487,A -85,B 0,C 180,E1 -8016.64,E2 -8016.64} C_VEL
LIN {X 0,Y 459.996,Z 606.559,A -85,B 0,C 180,E1 -8018.124,E2 -8018.124} C_VEL
LIN {X 0,Y 460.124,Z 598.744,A -85,B 0,C 180,E1 -8019.451,E2 -8019.451} C_VEL
LIN {X 0,Y 460.414,Z 589.074,A -85,B 0,C 180,E1 -8020.777,E2 -8020.777} C_VEL
LIN {X 0,Y 460.767,Z 580.181,A -85,B 0,C 180,E1 -8021.771,E2 -8021.771} C_VEL
LIN {X 0,Y 461.141,Z 569.146,A -85,B 0,C 180,E1 -8022.783,E2 -8022.783} C_VEL
LIN {X 0,Y 461.651,Z 557.361,A -85,B 0,C 180,E1 -8023.649,E2 -8023.649} C_VEL
LIN {X 0,Y 462.242,Z 544.766,A -85,B 0,C 180,E1 -8024.36,E2 -8024.36} C_VEL
LIN {X 0,Y 462.723,Z 530.992,A -85,B 0,C 180,E1 -8024.935,E2 -8024.935} C_VEL
LIN {X 0,Y 463.168,Z 518.282,A -85,B 0,C 180,E1 -8025.286,E2 -8025.286} C_VEL
LIN {X 0,Y 464.065,Z 435.755,A -85,B 0,C 180,E1 -8026.774,E2 -8026.774} C_VEL
LIN {X 0,Y 461.153,Z 407.789,A -85,B 0,C 180,E1 -8027.447,E2 -8027.447} C_VEL
LIN {X 0,Y 461.695,Z 389.329,A -85,B 0,C 180,E1 -8030.029,E2 -8030.029} C_VEL
LIN {X 0,Y 462.463,Z 371.5,A -85,B 0,C 180,E1 -8032.564,E2 -8032.564} C_VEL
LIN {X 0,Y 463.446,Z 350.697,A -85,B 0,C 180,E1 -8035.607,E2 -8035.607} C_VEL
LIN {X 0,Y 463.885,Z 339.656,A -85,B 0,C 180,E1 -8037.277,E2 -8037.277} C_VEL
LIN {X 0,Y 461.635,Z 328.746,A -85,B 0,C 180,E1 -8039.155,E2 -8039.155} C_VEL
LIN {X 0,Y 460.555,Z 324.121,A -85,B 0,C 180,E1 -8040.008,E2 -8040.008} C_VEL
LIN {X 0,Y 460.522,Z 324.122,A -85,B 0,C 180,E1 -8043.325,E2 -8043.325} C_VEL
LIN {X 0,Y 460.475,Z 324.129,A -85,B 0,C 180,E1 -8046.53,E2 -8046.53} C_VEL
LIN {X 0,Y 460.516,Z 324.124,A -85,B 0,C 180,E1 -8049.864,E2 -8049.864} C_VEL
LIN {X 0,Y 460.481,Z 324.125,A -85,B 0,C 180,E1 -8052.896,E2 -8052.896} C_VEL
LIN {X 0,Y 460.506,Z 324.125,A -85,B 0,C 180,E1 -8055.831,E2 -8055.831} C_VEL
LIN {X 0,Y 460.518,Z 324.119,A -85,B 0,C 180,E1 -8058.987,E2 -8058.987} C_VEL
LIN {X 0,Y 460.485,Z 324.125,A -85,B 0,C 180,E1 -8062.375,E2 -8062.375} C_VEL
LIN {X 0,Y 460.536,Z 324.12,A -85,B 0,C 180,E1 -8065.622,E2 -8065.622} C_VEL
LIN {X 0,Y 460.506,Z 324.121,A -85,B 0,C 180,E1 -8068.742,E2 -8068.742} C_VEL
LIN {X 0,Y 460.505,Z 324.125,A -85,B 0,C 180,E1 -8071.763,E2 -8071.763} C_VEL
LIN {X 0,Y 460.512,Z 324.121,A -85,B 0,C 180,E1 -8074.702,E2 -8074.702} C_VEL
LIN {X 0,Y 460.496,Z 324.128,A -85,B 0,C 180,E1 -8077.57,E2 -8077.57} C_VEL
LIN {X 0,Y 460.52,Z 324.121,A -85,B 0,C 180,E1 -8080.382,E2 -8080.382} C_VEL
LIN {X 0,Y 460.549,Z 324.12,A -85,B 0,C 180,E1 -8083.145,E2 -8083.145} C_VEL
LIN {X 0,Y 460.557,Z 324.122,A -85,B 0,C 180,E1 -8084.922,E2 -8084.922} C_VEL
LIN {X 0,Y 463.045,Z 330.822,A -85,B 0,C 180,E1 -8085.179,E2 -8085.179} C_VEL
LIN {X 0,Y 464.795,Z 335.505,A -85,B 0,C 180,E1 -8085.354,E2 -8085.354} C_VEL
LIN {X 0,Y 463.615,Z 415.731,A -85,B 0,C 180,E1 -8086.856,E2 -8086.856} C_VEL
LIN {X 0,Y 463.513,Z 429.283,A -85,B 0,C 180,E1 -8087.299,E2 -8087.299} C_VEL
LIN {X 0,Y 463.281,Z 441.003,A -85,B 0,C 180,E1 -8087.849,E2 -8087.849} C_VEL
LIN {X 0,Y 463.007,Z 453.197,A -85,B 0,C 180,E1 -8088.619,E2 -8088.619} C_VEL
LIN {X 0,Y 462.523,Z 464.16,A -85,B 0,C 180,E1 -8089.494,E2 -8089.494} C_VEL
LIN {X 0,Y 462.233,Z 473.007,A -85,B 0,C 180,E1 -8090.372,E2 -8090.372} C_VEL
LIN {X 0,Y 461.741,Z 482.057,A -85,B 0,C 180,E1 -8091.46,E2 -8091.46} C_VEL
LIN {X 0,Y 461.315,Z 490.895,A -85,B 0,C 180,E1 -8092.786,E2 -8092.786} C_VEL
LIN {X 0,Y 461.063,Z 497.868,A -85,B 0,C 180,E1 -8094.094,E2 -8094.094} C_VEL
LIN {X 0,Y 460.753,Z 502.594,A -85,B 0,C 180,E1 -8095.187,E2 -8095.187} C_VEL
LIN {X 0,Y 460.421,Z 507.154,A -85,B 0,C 180,E1 -8096.499,E2 -8096.499} C_VEL
LIN {X 0,Y 460.249,Z 509.565,A -85,B 0,C 180,E1 -8097.374,E2 -8097.374} C_VEL
LIN {X 0,Y 460.296,Z 511.464,A -85,B 0,C 180,E1 -8098.25,E2 -8098.25} C_VEL
LIN {X 0,Y 460.202,Z 512.97,A -85,B 0,C 180,E1 -8099.125,E2 -8099.125} C_VEL
LIN {X 0,Y 460.165,Z 514.052,A -85,B 0,C 180,E1 -8100,E2 -8100} C_VEL
LIN {X 0,Y 460.163,Z 514.681,A -85,B 0,C 180,E1 -8100.875,E2 -8100.875} C_VEL
LIN {X 0,Y 459.968,Z 514.945,A -85,B 0,C 180,E1 -8101.751,E2 -8101.751} C_VEL
LIN {X 0,Y 459.999,Z 514.79,A -85,B 0,C 180,E1 -8102.627,E2 -8102.627} C_VEL
LIN {X 0,Y 460.063,Z 514.208,A -85,B 0,C 180,E1 -8103.503,E2 -8103.503} C_VEL
LIN {X 0,Y 460.157,Z 513.198,A -85,B 0,C 180,E1 -8104.379,E2 -8104.379} C_VEL
LIN {X 0,Y 460.189,Z 511.798,A -85,B 0,C 180,E1 -8105.257,E2 -8105.257} C_VEL
LIN {X 0,Y 460.281,Z 508.468,A -85,B 0,C 180,E1 -8106.734,E2 -8106.734} C_VEL
LIN {X 0,Y 460.439,Z 504.881,A -85,B 0,C 180,E1 -8107.895,E2 -8107.895} C_VEL
LIN {X 0,Y 460.697,Z 498.738,A -85,B 0,C 180,E1 -8109.438,E2 -8109.438} C_VEL
LIN {X 0,Y 460.983,Z 491.965,A -85,B 0,C 180,E1 -8110.763,E2 -8110.763} C_VEL
LIN {X 0,Y 461.341,Z 483.54,A -85,B 0,C 180,E1 -8112.091,E2 -8112.091} C_VEL
LIN {X 0,Y 461.654,Z 474.862,A -85,B 0,C 180,E1 -8113.2,E2 -8113.2} C_VEL
LIN {X 0,Y 462.11,Z 464.102,A -85,B 0,C 180,E1 -8114.308,E2 -8114.308} C_VEL
LIN {X 0,Y 462.475,Z 453.412,A -85,B 0,C 180,E1 -8115.197,E2 -8115.197} C_VEL
LIN {X 0,Y 462.893,Z 441.519,A -85,B 0,C 180,E1 -8115.973,E2 -8115.973} C_VEL
LIN {X 0,Y 463.178,Z 429.178,A -85,B 0,C 180,E1 -8116.585,E2 -8116.585} C_VEL
LIN {X 0,Y 463.264,Z 415.741,A -85,B 0,C 180,E1 -8117.062,E2 -8117.062} C_VEL
LIN {X 0,Y 463.437,Z 398.803,A -85,B 0,C 180,E1 -8117.407,E2 -8117.407} C_VEL
LIN {X 0,Y 464.126,Z 334.662,A -85,B 0,C 180,E1 -8118.518,E2 -8118.518} C_VEL
LIN {X 0,Y 460.568,Z 324.118,A -85,B 0,C 180,E1 -8118.838,E2 -8118.838} C_VEL
LIN {X 0,Y 460.517,Z 324.118,A -85,B 0,C 180,E1 -8121.485,E2 -8121.485} C_VEL
LIN {X 0,Y 460.539,Z 324.117,A -85,B 0,C 180,E1 -8124.332,E2 -8124.332} C_VEL
LIN {X 0,Y 460.573,Z 324.112,A -85,B 0,C 180,E1 -8127.243,E2 -8127.243} C_VEL
LIN {X 0,Y 460.51,Z 324.121,A -85,B 0,C 180,E1 -8130.24,E2 -8130.24} C_VEL
LIN {X 0,Y 460.519,Z 324.118,A -85,B 0,C 180,E1 -8133.325,E2 -8133.325} C_VEL
LIN {X 0,Y 460.475,Z 324.128,A -85,B 0,C 180,E1 -8136.529,E2 -8136.529} C_VEL
LIN {X 0,Y 460.524,Z 324.118,A -85,B 0,C 180,E1 -8139.863,E2 -8139.863} C_VEL
LIN {X 0,Y 460.511,Z 324.121,A -85,B 0,C 180,E1 -8142.9,E2 -8142.9} C_VEL
LIN {X 0,Y 460.507,Z 324.12,A -85,B 0,C 180,E1 -8145.83,E2 -8145.83} C_VEL
LIN {X 0,Y 460.529,Z 324.118,A -85,B 0,C 180,E1 -8148.988,E2 -8148.988} C_VEL
LIN {X 0,Y 460.525,Z 324.117,A -85,B 0,C 180,E1 -8151.267,E2 -8151.267} C_VEL
LIN {X 0,Y 460.511,Z 324.124,A -85,B 0,C 180,E1 -8154.554,E2 -8154.554} C_VEL
LIN {X 0,Y 460.529,Z 324.118,A -85,B 0,C 180,E1 -8157.715,E2 -8157.715} C_VEL
LIN {X 0,Y 460.538,Z 324.118,A -85,B 0,C 180,E1 -8160.769,E2 -8160.769} C_VEL
LIN {X 0,Y 460.561,Z 324.114,A -85,B 0,C 180,E1 -8163.735,E2 -8163.735} C_VEL
LIN {X 0,Y 460.544,Z 324.118,A -85,B 0,C 180,E1 -8166.624,E2 -8166.624} C_VEL
LIN {X 0,Y 460.506,Z 324.12,A -85,B 0,C 180,E1 -8167.4,E2 -8167.4} C_VEL
LIN {X 0,Y 459.856,Z 324.206,A -85,B 0,C 180,E1 -8168.13,E2 -8168.13} C_VEL
LIN {X 0,Y 457.035,Z 324.555,A -85,B 0,C 180,E1 -8169.316,E2 -8169.316} C_VEL
LIN {X 0,Y 454.635,Z 324.856,A -85,B 0,C 180,E1 -8170.273,E2 -8170.273} C_VEL
LIN {X 0,Y 453.594,Z 324.981,A -85,B 0,C 180,E1 -8171.012,E2 -8171.012} C_VEL
LIN {X 0,Y 453.505,Z 324.991,A -85,B 0,C 180,E1 -8171.262,E2 -8171.262} C_VEL
LIN {X 0,Y 453.537,Z 324.989,A -85,B 0,C 180,E1 -8174.726,E2 -8174.726} C_VEL
LIN {X 0,Y 453.557,Z 324.99,A -85,B 0,C 180,E1 -8178.379,E2 -8178.379} C_VEL
LIN {X 0,Y 453.649,Z 324.977,A -85,B 0,C 180,E1 -8181.985,E2 -8181.985} C_VEL
LIN {X 0,Y 453.668,Z 324.973,A -85,B 0,C 180,E1 -8184.667,E2 -8184.667} C_VEL
LIN {X 0,Y 453.763,Z 324.96,A -85,B 0,C 180,E1 -8187.337,E2 -8187.337} C_VEL
LIN {X 0,Y 453.822,Z 324.957,A -85,B 0,C 180,E1 -8190,E2 -8190} C_VEL
LIN {X 0,Y 453.763,Z 324.961,A -85,B 0,C 180,E1 -8192.663,E2 -8192.663} C_VEL
LIN {X 0,Y 453.675,Z 324.975,A -85,B 0,C 180,E1 -8196.226,E2 -8196.226} C_VEL
LIN {X 0,Y 453.59,Z 324.981,A -85,B 0,C 180,E1 -8198.914,E2 -8198.914} C_VEL
LIN {X 0,Y 453.561,Z 324.986,A -85,B 0,C 180,E1 -8202.529,E2 -8202.529} C_VEL
LIN {X 0,Y 453.543,Z 324.991,A -85,B 0,C 180,E1 -8206.196,E2 -8206.196} C_VEL
LIN {X 0,Y 453.518,Z 324.991,A -85,B 0,C 180,E1 -8209.041,E2 -8209.041} C_VEL
LIN {X 0,Y 453.475,Z 325,A -85,B 0,C 180,E1 -8211.836,E2 -8211.836} C_VEL
LIN {X 0,Y 453.513,Z 324.991,A -85,B 0,C 180,E1 -8214.735,E2 -8214.735} C_VEL
LIN {X 0,Y 453.536,Z 324.993,A -85,B 0,C 180,E1 -8217.961,E2 -8217.961} C_VEL
LIN {X 0,Y 453.465,Z 324.999,A -85,B 0,C 180,E1 -8221.526,E2 -8221.526} C_VEL
LIN {X 0,Y 453.488,Z 324.994,A -85,B 0,C 180,E1 -8224.778,E2 -8224.778} C_VEL
LIN {X 0,Y 453.473,Z 324.997,A -85,B 0,C 180,E1 -8228.311,E2 -8228.311} C_VEL
LIN {X 0,Y 453.494,Z 324.994,A -85,B 0,C 180,E1 -8230.61,E2 -8230.61} C_VEL
LIN {X 0,Y 453.454,Z 325,A -85,B 0,C 180,E1 -8233.245,E2 -8233.245} C_VEL
LIN {X 0,Y 453.464,Z 325.003,A -85,B 0,C 180,E1 -8235.779,E2 -8235.779} C_VEL
LIN {X 0,Y 453.479,Z 324.996,A -85,B 0,C 180,E1 -8238.21,E2 -8238.21} C_VEL
LIN {X 0,Y 453.488,Z 324.995,A -85,B 0,C 180,E1 -8240.795,E2 -8240.795} C_VEL
LIN {X 0,Y 453.455,Z 325.001,A -85,B 0,C 180,E1 -8243.918,E2 -8243.918} C_VEL
LIN {X 0,Y 453.48,Z 324.997,A -85,B 0,C 180,E1 -8247.152,E2 -8247.152} C_VEL
LIN {X 0,Y 453.476,Z 324.996,A -85,B 0,C 180,E1 -8250.269,E2 -8250.269} C_VEL
LIN {X 0,Y 453.507,Z 324.996,A -85,B 0,C 180,E1 -8253.294,E2 -8253.294} C_VEL
LIN {X 0,Y 453.509,Z 325.01,A -85,B 0,C 180,E1 -8255.024,E2 -8255.024} C_VEL
LIN {X 0,Y 457.335,Z 336.466,A -85,B 0,C 180,E1 -8255.369,E2 -8255.369} C_VEL
LIN {X 0,Y 456.485,Z 413.327,A -85,B 0,C 180,E1 -8256.734,E2 -8256.734} C_VEL
LIN {X 0,Y 456.354,Z 425.535,A -85,B 0,C 180,E1 -8257.117,E2 -8257.117} C_VEL
LIN {X 0,Y 456.084,Z 437.733,A -85,B 0,C 180,E1 -8257.669,E2 -8257.669} C_VEL
LIN {X 0,Y 455.754,Z 449.826,A -85,B 0,C 180,E1 -8258.398,E2 -8258.398} C_VEL
LIN {X 0,Y 455.367,Z 460.403,A -85,B 0,C 180,E1 -8259.209,E2 -8259.209} C_VEL
LIN {X 0,Y 454.942,Z 471.296,A -85,B 0,C 180,E1 -8260.259,E2 -8260.259} C_VEL
LIN {X 0,Y 454.513,Z 480.036,A -85,B 0,C 180,E1 -8261.286,E2 -8261.286} C_VEL
LIN {X 0,Y 454.164,Z 488.124,A -85,B 0,C 180,E1 -8262.437,E2 -8262.437} C_VEL
LIN {X 0,Y 453.769,Z 495.92,A -85,B 0,C 180,E1 -8263.813,E2 -8263.813} C_VEL
LIN {X 0,Y 453.512,Z 502.132,A -85,B 0,C 180,E1 -8265.186,E2 -8265.186} C_VEL
LIN {X 0,Y 453.314,Z 507.005,A -85,B 0,C 180,E1 -8266.553,E2 -8266.553} C_VEL
LIN {X 0,Y 453.247,Z 510.048,A -85,B 0,C 180,E1 -8267.656,E2 -8267.656} C_VEL
LIN {X 0,Y 453.04,Z 513.315,A -85,B 0,C 180,E1 -8269.272,E2 -8269.272} C_VEL
LIN {X 0,Y 453.034,Z 514.491,A -85,B 0,C 180,E1 -8270.175,E2 -8270.175} C_VEL
LIN {X 0,Y 453.056,Z 515.245,A -85,B 0,C 180,E1 -8271.076,E2 -8271.076} C_VEL
LIN {X 0,Y 453.077,Z 515.606,A -85,B 0,C 180,E1 -8271.975,E2 -8271.975} C_VEL
LIN {X 0,Y 453.137,Z 515.455,A -85,B 0,C 180,E1 -8273.038,E2 -8273.038} C_VEL
LIN {X 0,Y 453.202,Z 514.132,A -85,B 0,C 180,E1 -8274.662,E2 -8274.662} C_VEL
LIN {X 0,Y 453.207,Z 512.827,A -85,B 0,C 180,E1 -8275.553,E2 -8275.553} C_VEL
LIN {X 0,Y 453.334,Z 510.027,A -85,B 0,C 180,E1 -8276.89,E2 -8276.89} C_VEL
LIN {X 0,Y 453.566,Z 506.171,A -85,B 0,C 180,E1 -8278.225,E2 -8278.225} C_VEL
LIN {X 0,Y 453.851,Z 501.156,A -85,B 0,C 180,E1 -8279.557,E2 -8279.557} C_VEL
LIN {X 0,Y 454.252,Z 494.82,A -85,B 0,C 180,E1 -8280.887,E2 -8280.887} C_VEL
LIN {X 0,Y 454.67,Z 486.958,A -85,B 0,C 180,E1 -8282.215,E2 -8282.215} C_VEL
LIN {X 0,Y 455.094,Z 478.85,A -85,B 0,C 180,E1 -8283.32,E2 -8283.32} C_VEL
LIN {X 0,Y 455.535,Z 468.904,A -85,B 0,C 180,E1 -8284.425,E2 -8284.425} C_VEL
LIN {X 0,Y 455.955,Z 457.76,A -85,B 0,C 180,E1 -8285.418,E2 -8285.418} C_VEL
LIN {X 0,Y 456.373,Z 446.669,A -85,B 0,C 180,E1 -8286.189,E2 -8286.189} C_VEL
LIN {X 0,Y 456.649,Z 434.376,A -85,B 0,C 180,E1 -8286.851,E2 -8286.851} C_VEL
LIN {X 0,Y 456.8,Z 421.38,A -85,B 0,C 180,E1 -8287.348,E2 -8287.348} C_VEL
LIN {X 0,Y 456.903,Z 407.505,A -85,B 0,C 180,E1 -8287.68,E2 -8287.68} C_VEL
LIN {X 0,Y 457.922,Z 336.592,A -85,B 0,C 180,E1 -8288.989,E2 -8288.989} C_VEL
LIN {X 0,Y 453.591,Z 325.367,A -85,B 0,C 180,E1 -8289.421,E2 -8289.421} C_VEL
LIN {X 0,Y 453.543,Z 324.993,A -85,B 0,C 180,E1 -8289.46,E2 -8289.46} C_VEL
LIN {X 0,Y 453.569,Z 324.99,A -85,B 0,C 180,E1 -8292.529,E2 -8292.529} C_VEL
LIN {X 0,Y 453.542,Z 324.993,A -85,B 0,C 180,E1 -8296.196,E2 -8296.196} C_VEL
LIN {X 0,Y 453.49,Z 324.999,A -85,B 0,C 180,E1 -8299.028,E2 -8299.028} C_VEL
LIN {X 0,Y 453.472,Z 325.001,A -85,B 0,C 180,E1 -8301.837,E2 -8301.837} C_VEL
LIN {X 0,Y 453.465,Z 325.001,A -85,B 0,C 180,E1 -8304.738,E2 -8304.738} C_VEL
LIN {X 0,Y 453.463,Z 325.001,A -85,B 0,C 180,E1 -8307.942,E2 -8307.942} C_VEL
LIN {X 0,Y 453.459,Z 324.999,A -85,B 0,C 180,E1 -8310.761,E2 -8310.761} C_VEL
LIN {X 0,Y 453.469,Z 324.999,A -85,B 0,C 180,E1 -8313.914,E2 -8313.914} C_VEL
LIN {X 0,Y 453.439,Z 324.998,A -85,B 0,C 180,E1 -8317.191,E2 -8317.191} C_VEL
LIN {X 0,Y 453.474,Z 324.994,A -85,B 0,C 180,E1 -8320.612,E2 -8320.612} C_VEL
LIN {X 0,Y 453.485,Z 324.995,A -85,B 0,C 180,E1 -8324.528,E2 -8324.528} C_VEL
LIN {X 0,Y 453.452,Z 325.002,A -85,B 0,C 180,E1 -8328.069,E2 -8328.069} C_VEL
LIN {X 0,Y 453.451,Z 324.999,A -85,B 0,C 180,E1 -8330.801,E2 -8330.801} C_VEL
LIN {X 0,Y 453.454,Z 325.002,A -85,B 0,C 180,E1 -8333.917,E2 -8333.917} C_VEL
LIN {X 0,Y 453.483,Z 324.998,A -85,B 0,C 180,E1 -8337.151,E2 -8337.151} C_VEL
LIN {X 0,Y 453.508,Z 325.142,A -85,B 0,C 180,E1 -8339.731,E2 -8339.731} C_VEL
LIN {X 0,Y 456.985,Z 340.841,A -85,B 0,C 180,E1 -8342.275,E2 -8342.275} C_VEL
LIN {X 0,Y 457.397,Z 344.62,A -85,B 0,C 180,E1 -8342.858,E2 -8342.858} C_VEL
LIN {X 0,Y 456.208,Z 367.29,A -85,B 0,C 180,E1 -8346.147,E2 -8346.147} C_VEL
LIN {X 0,Y 455.214,Z 388.605,A -85,B 0,C 180,E1 -8349.2,E2 -8349.2} C_VEL
LIN {X 0,Y 454.478,Z 408.205,A -85,B 0,C 180,E1 -8351.984,E2 -8351.984} C_VEL
LIN {X 0,Y 454.348,Z 411.982,A -85,B 0,C 180,E1 -8352.517,E2 -8352.517} C_VEL
LIN {X 0,Y 457.162,Z 438.894,A -85,B 0,C 180,E1 -8353.11,E2 -8353.11} C_VEL
LIN {X 0,Y 456.124,Z 522.555,A -85,B 0,C 180,E1 -8354.614,E2 -8354.614} C_VEL
LIN {X 0,Y 455.594,Z 536.627,A -85,B 0,C 180,E1 -8355.054,E2 -8355.054} C_VEL
LIN {X 0,Y 455.15,Z 549.23,A -85,B 0,C 180,E1 -8355.639,E2 -8355.639} C_VEL
LIN {X 0,Y 454.528,Z 560.912,A -85,B 0,C 180,E1 -8356.361,E2 -8356.361} C_VEL
LIN {X 0,Y 454.082,Z 571.423,A -85,B 0,C 180,E1 -8357.182,E2 -8357.182} C_VEL
LIN {X 0,Y 453.805,Z 580.478,A -85,B 0,C 180,E1 -8358.045,E2 -8358.045} C_VEL
LIN {X 0,Y 453.419,Z 589.298,A -85,B 0,C 180,E1 -8359.054,E2 -8359.054} C_VEL
LIN {X 0,Y 453.056,Z 597.423,A -85,B 0,C 180,E1 -8360.175,E2 -8360.175} C_VEL
LIN {X 0,Y 452.895,Z 605.375,A -85,B 0,C 180,E1 -8361.522,E2 -8361.522} C_VEL
LIN {X 0,Y 452.764,Z 611.722,A -85,B 0,C 180,E1 -8362.866,E2 -8362.866} C_VEL
LIN {X 0,Y 452.769,Z 616.747,A -85,B 0,C 180,E1 -8364.209,E2 -8364.209} C_VEL
LIN {X 0,Y 452.82,Z 620.583,A -85,B 0,C 180,E1 -8365.549,E2 -8365.549} C_VEL
LIN {X 0,Y 452.881,Z 622.546,A -85,B 0,C 180,E1 -8366.441,E2 -8366.441} C_VEL
LIN {X 0,Y 452.781,Z 624.025,A -85,B 0,C 180,E1 -8367.331,E2 -8367.331} C_VEL
LIN {X 0,Y 452.756,Z 625.04,A -85,B 0,C 180,E1 -8368.221,E2 -8368.221} C_VEL
LIN {X 0,Y 452.765,Z 625.643,A -85,B 0,C 180,E1 -8369.11,E2 -8369.11} C_VEL
LIN {X 0,Y 452.79,Z 625.831,A -85,B 0,C 180,E1 -8370,E2 -8370} C_VEL
LIN {X 0,Y 452.775,Z 625.557,A -85,B 0,C 180,E1 -8370.889,E2 -8370.889} C_VEL
LIN {X 0,Y 452.776,Z 624.846,A -85,B 0,C 180,E1 -8371.779,E2 -8371.779} C_VEL
LIN {X 0,Y 452.803,Z 623.72,A -85,B 0,C 180,E1 -8372.669,E2 -8372.669} C_VEL
LIN {X 0,Y 452.888,Z 621.184,A -85,B 0,C 180,E1 -8374.004,E2 -8374.004} C_VEL
LIN {X 0,Y 452.77,Z 617.56,A -85,B 0,C 180,E1 -8375.344,E2 -8375.344} C_VEL
LIN {X 0,Y 452.829,Z 612.988,A -85,B 0,C 180,E1 -8376.637,E2 -8376.637} C_VEL
LIN {X 0,Y 452.887,Z 606.773,A -85,B 0,C 180,E1 -8378.028,E2 -8378.028} C_VEL
LIN {X 0,Y 453.015,Z 599.238,A -85,B 0,C 180,E1 -8379.375,E2 -8379.375} C_VEL
LIN {X 0,Y 453.303,Z 589.854,A -85,B 0,C 180,E1 -8380.722,E2 -8380.722} C_VEL
LIN {X 0,Y 453.706,Z 580.275,A -85,B 0,C 180,E1 -8381.844,E2 -8381.844} C_VEL
LIN {X 0,Y 454.118,Z 569.157,A -85,B 0,C 180,E1 -8382.9,E2 -8382.9} C_VEL
LIN {X 0,Y 454.625,Z 558.036,A -85,B 0,C 180,E1 -8383.75,E2 -8383.75} C_VEL
LIN {X 0,Y 455.199,Z 546.054,A -85,B 0,C 180,E1 -8384.473,E2 -8384.473} C_VEL
LIN {X 0,Y 455.765,Z 532.408,A -85,B 0,C 180,E1 -8385.083,E2 -8385.083} C_VEL
LIN {X 0,Y 456.298,Z 518.874,A -85,B 0,C 180,E1 -8385.494,E2 -8385.494} C_VEL
LIN {X 0,Y 457.234,Z 436.035,A -85,B 0,C 180,E1 -8387.044,E2 -8387.044} C_VEL
LIN {X 0,Y 454.431,Z 408.888,A -85,B 0,C 180,E1 -8387.714,E2 -8387.714} C_VEL
LIN {X 0,Y 454.146,Z 406.676,A -85,B 0,C 180,E1 -8387.773,E2 -8387.773} C_VEL
LIN {X 0,Y 454.877,Z 387.025,A -85,B 0,C 180,E1 -8390.579,E2 -8390.579} C_VEL
LIN {X 0,Y 455.839,Z 366.127,A -85,B 0,C 180,E1 -8393.632,E2 -8393.632} C_VEL
LIN {X 0,Y 457.129,Z 343.27,A -85,B 0,C 180,E1 -8397.099,E2 -8397.099} C_VEL
LIN {X 0,Y 456.45,Z 337.84,A -85,B 0,C 180,E1 -8398.009,E2 -8398.009} C_VEL
LIN {X 0,Y 453.623,Z 325.578,A -85,B 0,C 180,E1 -8400.251,E2 -8400.251} C_VEL
LIN {X 0,Y 453.498,Z 325.001,A -85,B 0,C 180,E1 -8400.384,E2 -8400.384} C_VEL
LIN {X 0,Y 453.471,Z 325.001,A -85,B 0,C 180,E1 -8403.913,E2 -8403.913} C_VEL
LIN {X 0,Y 453.452,Z 325,A -85,B 0,C 180,E1 -8407.19,E2 -8407.19} C_VEL
LIN {X 0,Y 453.473,Z 325.001,A -85,B 0,C 180,E1 -8410.611,E2 -8410.611} C_VEL
LIN {X 0,Y 453.461,Z 325.004,A -85,B 0,C 180,E1 -8414.222,E2 -8414.222} C_VEL
LIN {X 0,Y 453.439,Z 325,A -85,B 0,C 180,E1 -8417.002,E2 -8417.002} C_VEL
LIN {X 0,Y 453.472,Z 324.998,A -85,B 0,C 180,E1 -8419.412,E2 -8419.412} C_VEL
LIN {X 0,Y 453.437,Z 325,A -85,B 0,C 180,E1 -8422.808,E2 -8422.808} C_VEL
LIN {X 0,Y 453.467,Z 325.001,A -85,B 0,C 180,E1 -8426.086,E2 -8426.086} C_VEL
LIN {X 0,Y 453.457,Z 325.001,A -85,B 0,C 180,E1 -8429.239,E2 -8429.239} C_VEL
LIN {X 0,Y 453.473,Z 324.999,A -85,B 0,C 180,E1 -8432.293,E2 -8432.293} C_VEL
LIN {X 0,Y 453.463,Z 325.002,A -85,B 0,C 180,E1 -8435.262,E2 -8435.262} C_VEL
LIN {X 0,Y 453.478,Z 324.999,A -85,B 0,C 180,E1 -8438.417,E2 -8438.417} C_VEL
LIN {X 0,Y 453.488,Z 324.998,A -85,B 0,C 180,E1 -8441.007,E2 -8441.007} C_VEL
LIN {X 0,Y 453.566,Z 324.99,A -85,B 0,C 180,E1 -8444.571,E2 -8444.571} C_VEL
LIN {X 0,Y 455.982,Z 331.533,A -85,B 0,C 180,E1 -8444.85,E2 -8444.85} C_VEL
LIN {X 0,Y 458.145,Z 337.12,A -85,B 0,C 180,E1 -8445.073,E2 -8445.073} C_VEL
LIN {X 0,Y 456.852,Z 416.544,A -85,B 0,C 180,E1 -8446.604,E2 -8446.604} C_VEL
LIN {X 0,Y 456.736,Z 430.016,A -85,B 0,C 180,E1 -8447.051,E2 -8447.051} C_VEL
LIN {X 0,Y 456.486,Z 442.747,A -85,B 0,C 180,E1 -8447.665,E2 -8447.665} C_VEL
LIN {X 0,Y 456.195,Z 454.783,A -85,B 0,C 180,E1 -8448.447,E2 -8448.447} C_VEL
LIN {X 0,Y 455.669,Z 465.622,A -85,B 0,C 180,E1 -8449.334,E2 -8449.334} C_VEL
LIN {X 0,Y 455.194,Z 476.3,A -85,B 0,C 180,E1 -8450.446,E2 -8450.446} C_VEL
LIN {X 0,Y 454.808,Z 484.421,A -85,B 0,C 180,E1 -8451.484,E2 -8451.484} C_VEL
LIN {X 0,Y 454.374,Z 492.069,A -85,B 0,C 180,E1 -8452.668,E2 -8452.668} C_VEL
LIN {X 0,Y 454.086,Z 499.031,A -85,B 0,C 180,E1 -8454.003,E2 -8454.003} C_VEL
LIN {X 0,Y 453.771,Z 503.715,A -85,B 0,C 180,E1 -8455.113,E2 -8455.113} C_VEL
LIN {X 0,Y 453.417,Z 508.23,A -85,B 0,C 180,E1 -8456.445,E2 -8456.445} C_VEL
LIN {X 0,Y 453.259,Z 510.595,A -85,B 0,C 180,E1 -8457.333,E2 -8457.333} C_VEL
LIN {X 0,Y 453.298,Z 512.47,A -85,B 0,C 180,E1 -8458.223,E2 -8458.223} C_VEL
LIN {X 0,Y 453.177,Z 513.954,A -85,B 0,C 180,E1 -8459.111,E2 -8459.111} C_VEL
LIN {X 0,Y 453.138,Z 514.996,A -85,B 0,C 180,E1 -8460,E2 -8460} C_VEL
LIN {X 0,Y 453.132,Z 515.6,A -85,B 0,C 180,E1 -8460.888,E2 -8460.888} C_VEL
LIN {X 0,Y 452.925,Z 515.838,A -85,B 0,C 180,E1 -8461.778,E2 -8461.778} C_VEL
LIN {X 0,Y 452.956,Z 515.653,A -85,B 0,C 180,E1 -8462.668,E2 -8462.668} C_VEL
LIN {X 0,Y 453.019,Z 515.022,A -85,B 0,C 180,E1 -8463.557,E2 -8463.557} C_VEL
LIN {X 0,Y 453.13,Z 513.979,A -85,B 0,C 180,E1 -8464.447,E2 -8464.447} C_VEL
LIN {X 0,Y 453.165,Z 512.543,A -85,B 0,C 180,E1 -8465.339,E2 -8465.339} C_VEL
LIN {X 0,Y 453.283,Z 508.869,A -85,B 0,C 180,E1 -8466.927,E2 -8466.927} C_VEL
LIN {X 0,Y 453.484,Z 503.865,A -85,B 0,C 180,E1 -8468.466,E2 -8468.466} C_VEL
LIN {X 0,Y 453.734,Z 498.186,A -85,B 0,C 180,E1 -8469.81,E2 -8469.81} C_VEL
LIN {X 0,Y 454.05,Z 491.085,A -85,B 0,C 180,E1 -8471.156,E2 -8471.156} C_VEL
LIN {X 0,Y 454.428,Z 482.147,A -85,B 0,C 180,E1 -8472.504,E2 -8472.504} C_VEL
LIN {X 0,Y 454.849,Z 471.958,A -85,B 0,C 180,E1 -8473.742,E2 -8473.742} C_VEL
LIN {X 0,Y 455.316,Z 461.508,A -85,B 0,C 180,E1 -8474.754,E2 -8474.754} C_VEL
LIN {X 0,Y 455.663,Z 449.896,A -85,B 0,C 180,E1 -8475.659,E2 -8475.659} C_VEL
LIN {X 0,Y 456.113,Z 437.766,A -85,B 0,C 180,E1 -8476.389,E2 -8476.389} C_VEL
LIN {X 0,Y 456.34,Z 424.332,A -85,B 0,C 180,E1 -8476.985,E2 -8476.985} C_VEL
LIN {X 0,Y 456.458,Z 411.808,A -85,B 0,C 180,E1 -8477.365,E2 -8477.365} C_VEL
LIN {X 0,Y 457.183,Z 335.903,A -85,B 0,C 180,E1 -8478.729,E2 -8478.729} C_VEL
LIN {X 0,Y 453.527,Z 324.993,A -85,B 0,C 180,E1 -8479.082,E2 -8479.082} C_VEL
LIN {X 0,Y 453.477,Z 324.995,A -85,B 0,C 180,E1 -8481.836,E2 -8481.836} C_VEL
LIN {X 0,Y 453.508,Z 324.998,A -85,B 0,C 180,E1 -8484.734,E2 -8484.734} C_VEL
LIN {X 0,Y 453.533,Z 324.989,A -85,B 0,C 180,E1 -8487.959,E2 -8487.959} C_VEL
LIN {X 0,Y 453.465,Z 324.996,A -85,B 0,C 180,E1 -8491.524,E2 -8491.524} C_VEL
LIN {X 0,Y 453.482,Z 324.999,A -85,B 0,C 180,E1 -8494.776,E2 -8494.776} C_VEL
LIN {X 0,Y 453.459,Z 325,A -85,B 0,C 180,E1 -8498.312,E2 -8498.312} C_VEL
LIN {X 0,Y 453.492,Z 325,A -85,B 0,C 180,E1 -8500.608,E2 -8500.608} C_VEL
LIN {X 0,Y 453.453,Z 324.998,A -85,B 0,C 180,E1 -8503.244,E2 -8503.244} C_VEL
LIN {X 0,Y 453.462,Z 324.998,A -85,B 0,C 180,E1 -8505.778,E2 -8505.778} C_VEL
LIN {X 0,Y 453.477,Z 324.998,A -85,B 0,C 180,E1 -8508.209,E2 -8508.209} C_VEL
LIN {X 0,Y 453.513,Z 324.993,A -85,B 0,C 180,E1 -8510.79,E2 -8510.79} C_VEL
LIN {X 0,Y 453.455,Z 324.999,A -85,B 0,C 180,E1 -8513.917,E2 -8513.917} C_VEL
LIN {X 0,Y 453.481,Z 324.995,A -85,B 0,C 180,E1 -8517.151,E2 -8517.151} C_VEL
LIN {X 0,Y 453.473,Z 325,A -85,B 0,C 180,E1 -8520.268,E2 -8520.268} C_VEL
LIN {X 0,Y 453.507,Z 324.991,A -85,B 0,C 180,E1 -8523.294,E2 -8523.294} C_VEL
LIN {X 0,Y 453.501,Z 324.997,A -85,B 0,C 180,E1 -8526.239,E2 -8526.239} C_VEL
LIN {X 0,Y 453.48,Z 324.995,A -85,B 0,C 180,E1 -8529.118,E2 -8529.118} C_VEL
LIN {X 0,Y 453.505,Z 324.991,A -85,B 0,C 180,E1 -8531.262,E2 -8531.262} C_VEL
LIN {X 0,Y 452.826,Z 325.081,A -85,B 0,C 180,E1 -8532.004,E2 -8532.004} C_VEL
LIN {X 0,Y 449.976,Z 325.431,A -85,B 0,C 180,E1 -8533.209,E2 -8533.209} C_VEL
LIN {X 0,Y 447.575,Z 325.735,A -85,B 0,C 180,E1 -8534.181,E2 -8534.181} C_VEL
LIN {X 0,Y 446.548,Z 325.859,A -85,B 0,C 180,E1 -8534.932,E2 -8534.932} C_VEL
LIN {X 0,Y 446.466,Z 325.869,A -85,B 0,C 180,E1 -8535.187,E2 -8535.187} C_VEL
LIN {X 0,Y 446.515,Z 325.868,A -85,B 0,C 180,E1 -8538.193,E2 -8538.193} C_VEL
LIN {X 0,Y 446.598,Z 325.854,A -85,B 0,C 180,E1 -8541.858,E2 -8541.858} C_VEL
LIN {X 0,Y 446.643,Z 325.849,A -85,B 0,C 180,E1 -8544.583,E2 -8544.583} C_VEL
LIN {X 0,Y 446.707,Z 325.839,A -85,B 0,C 180,E1 -8547.295,E2 -8547.295} C_VEL
LIN {X 0,Y 446.792,Z 325.832,A -85,B 0,C 180,E1 -8550,E2 -8550} C_VEL
LIN {X 0,Y 446.706,Z 325.84,A -85,B 0,C 180,E1 -8552.705,E2 -8552.705} C_VEL
LIN {X 0,Y 446.644,Z 325.85,A -85,B 0,C 180,E1 -8556.324,E2 -8556.324} C_VEL
LIN {X 0,Y 446.536,Z 325.86,A -85,B 0,C 180,E1 -8559.056,E2 -8559.056} C_VEL
LIN {X 0,Y 446.519,Z 325.862,A -85,B 0,C 180,E1 -8562.73,E2 -8562.73} C_VEL
LIN {X 0,Y 446.494,Z 325.869,A -85,B 0,C 180,E1 -8566.228,E2 -8566.228} C_VEL
LIN {X 0,Y 446.467,Z 325.87,A -85,B 0,C 180,E1 -8569.304,E2 -8569.304} C_VEL
LIN {X 0,Y 446.417,Z 325.878,A -85,B 0,C 180,E1 -8572.2,E2 -8572.2} C_VEL
LIN {X 0,Y 446.457,Z 325.871,A -85,B 0,C 180,E1 -8575.153,E2 -8575.153} C_VEL
LIN {X 0,Y 446.483,Z 325.87,A -85,B 0,C 180,E1 -8578.179,E2 -8578.179} C_VEL
LIN {X 0,Y 446.418,Z 325.879,A -85,B 0,C 180,E1 -8581.776,E2 -8581.776} C_VEL
LIN {X 0,Y 446.429,Z 325.874,A -85,B 0,C 180,E1 -8584.523,E2 -8584.523} C_VEL
LIN {X 0,Y 446.43,Z 325.876,A -85,B 0,C 180,E1 -8588.082,E2 -8588.082} C_VEL
LIN {X 0,Y 446.427,Z 325.875,A -85,B 0,C 180,E1 -8590.918,E2 -8590.918} C_VEL
LIN {X 0,Y 446.4,Z 325.882,A -85,B 0,C 180,E1 -8593.847,E2 -8593.847} C_VEL
LIN {X 0,Y 446.398,Z 325.878,A -85,B 0,C 180,E1 -8596.404,E2 -8596.404} C_VEL
LIN {X 0,Y 446.427,Z 325.875,A -85,B 0,C 180,E1 -8599.083,E2 -8599.083} C_VEL
LIN {X 0,Y 446.408,Z 325.878,A -85,B 0,C 180,E1 -8602.122,E2 -8602.122} C_VEL
LIN {X 0,Y 446.424,Z 325.878,A -85,B 0,C 180,E1 -8605.477,E2 -8605.477} C_VEL
LIN {X 0,Y 446.417,Z 325.876,A -85,B 0,C 180,E1 -8608.7,E2 -8608.7} C_VEL
LIN {X 0,Y 446.487,Z 325.87,A -85,B 0,C 180,E1 -8611.822,E2 -8611.822} C_VEL
LIN {X 0,Y 446.485,Z 325.867,A -85,B 0,C 180,E1 -8614.78,E2 -8614.78} C_VEL
LIN {X 0,Y 450.491,Z 337.863,A -85,B 0,C 180,E1 -8615.154,E2 -8615.154} C_VEL
LIN {X 0,Y 449.606,Z 412.895,A -85,B 0,C 180,E1 -8616.51,E2 -8616.51} C_VEL
LIN {X 0,Y 449.462,Z 425.51,A -85,B 0,C 180,E1 -8616.898,E2 -8616.898} C_VEL
LIN {X 0,Y 449.228,Z 437.445,A -85,B 0,C 180,E1 -8617.433,E2 -8617.433} C_VEL
LIN {X 0,Y 448.856,Z 449.73,A -85,B 0,C 180,E1 -8618.17,E2 -8618.17} C_VEL
LIN {X 0,Y 448.443,Z 460.499,A -85,B 0,C 180,E1 -8618.993,E2 -8618.993} C_VEL
LIN {X 0,Y 448.044,Z 470.775,A -85,B 0,C 180,E1 -8619.974,E2 -8619.974} C_VEL
LIN {X 0,Y 447.528,Z 481.313,A -85,B 0,C 180,E1 -8621.221,E2 -8621.221} C_VEL
LIN {X 0,Y 447.146,Z 489.327,A -85,B 0,C 180,E1 -8622.389,E2 -8622.389} C_VEL
LIN {X 0,Y 446.771,Z 497.167,A -85,B 0,C 180,E1 -8623.809,E2 -8623.809} C_VEL
LIN {X 0,Y 446.456,Z 504.129,A -85,B 0,C 180,E1 -8625.412,E2 -8625.412} C_VEL
LIN {X 0,Y 446.251,Z 508.727,A -85,B 0,C 180,E1 -8626.8,E2 -8626.8} C_VEL
LIN {X 0,Y 446.154,Z 512.175,A -85,B 0,C 180,E1 -8628.184,E2 -8628.184} C_VEL
LIN {X 0,Y 446.013,Z 513.896,A -85,B 0,C 180,E1 -8629.101,E2 -8629.101} C_VEL
LIN {X 0,Y 446.007,Z 515.189,A -85,B 0,C 180,E1 -8630.019,E2 -8630.019} C_VEL
LIN {X 0,Y 446.002,Z 516.011,A -85,B 0,C 180,E1 -8630.934,E2 -8630.934} C_VEL
LIN {X 0,Y 446.022,Z 516.431,A -85,B 0,C 180,E1 -8631.848,E2 -8631.848} C_VEL
LIN {X 0,Y 446.111,Z 516.372,A -85,B 0,C 180,E1 -8632.981,E2 -8632.981} C_VEL
LIN {X 0,Y 446.159,Z 515.192,A -85,B 0,C 180,E1 -8634.577,E2 -8634.577} C_VEL
LIN {X 0,Y 446.176,Z 513.971,A -85,B 0,C 180,E1 -8635.483,E2 -8635.483} C_VEL
LIN {X 0,Y 446.306,Z 511.29,A -85,B 0,C 180,E1 -8636.841,E2 -8636.841} C_VEL
LIN {X 0,Y 446.578,Z 507.558,A -85,B 0,C 180,E1 -8638.197,E2 -8638.197} C_VEL
LIN {X 0,Y 446.886,Z 502.676,A -85,B 0,C 180,E1 -8639.55,E2 -8639.55} C_VEL
LIN {X 0,Y 447.29,Z 496.47,A -85,B 0,C 180,E1 -8640.901,E2 -8640.901} C_VEL
LIN {X 0,Y 447.698,Z 488.759,A -85,B 0,C 180,E1 -8642.25,E2 -8642.25} C_VEL
LIN {X 0,Y 448.167,Z 480.854,A -85,B 0,C 180,E1 -8643.372,E2 -8643.372} C_VEL
LIN {X 0,Y 448.634,Z 471.149,A -85,B 0,C 180,E1 -8644.493,E2 -8644.493} C_VEL
LIN {X 0,Y 449.059,Z 460.363,A -85,B 0,C 180,E1 -8645.501,E2 -8645.501} C_VEL
LIN {X 0,Y 449.526,Z 449.825,A -85,B 0,C 180,E1 -8646.283,E2 -8646.283} C_VEL
LIN {X 0,Y 449.873,Z 437.074,A -85,B 0,C 180,E1 -8647.011,E2 -8647.011} C_VEL
LIN {X 0,Y 450.072,Z 424.275,A -85,B 0,C 180,E1 -8647.543,E2 -8647.543} C_VEL
LIN {X 0,Y 450.158,Z 410.347,A -85,B 0,C 180,E1 -8647.908,E2 -8647.908} C_VEL
LIN {X 0,Y 451.305,Z 338.259,A -85,B 0,C 180,E1 -8649.27,E2 -8649.27} C_VEL
LIN {X 0,Y 446.601,Z 326.487,A -85,B 0,C 180,E1 -8649.754,E2 -8649.754} C_VEL
LIN {X 0,Y 446.494,Z 325.872,A -85,B 0,C 180,E1 -8649.799,E2 -8649.799} C_VEL
LIN {X 0,Y 446.526,Z 325.867,A -85,B 0,C 180,E1 -8652.73,E2 -8652.73} C_VEL
LIN {X 0,Y 446.487,Z 325.871,A -85,B 0,C 180,E1 -8656.46,E2 -8656.46} C_VEL
LIN {X 0,Y 446.431,Z 325.877,A -85,B 0,C 180,E1 -8659.305,E2 -8659.305} C_VEL
LIN {X 0,Y 446.41,Z 325.883,A -85,B 0,C 180,E1 -8662.2,E2 -8662.2} C_VEL
LIN {X 0,Y 446.416,Z 325.877,A -85,B 0,C 180,E1 -8665.155,E2 -8665.155} C_VEL
LIN {X 0,Y 446.42,Z 325.88,A -85,B 0,C 180,E1 -8668.184,E2 -8668.184} C_VEL
LIN {X 0,Y 446.411,Z 325.876,A -85,B 0,C 180,E1 -8671.301,E2 -8671.301} C_VEL
LIN {X 0,Y 446.424,Z 325.873,A -85,B 0,C 180,E1 -8674.524,E2 -8674.524} C_VEL
LIN {X 0,Y 446.402,Z 325.878,A -85,B 0,C 180,E1 -8678.076,E2 -8678.076} C_VEL
LIN {X 0,Y 446.404,Z 325.875,A -85,B 0,C 180,E1 -8681.394,E2 -8681.394} C_VEL
LIN {X 0,Y 446.425,Z 325.874,A -85,B 0,C 180,E1 -8685.108,E2 -8685.108} C_VEL
LIN {X 0,Y 446.41,Z 325.875,A -85,B 0,C 180,E1 -8688.606,E2 -8688.606} C_VEL
LIN {X 0,Y 446.413,Z 325.88,A -85,B 0,C 180,E1 -8691.922,E2 -8691.922} C_VEL
LIN {X 0,Y 446.426,Z 325.879,A -85,B 0,C 180,E1 -8695.476,E2 -8695.476} C_VEL
LIN {X 0,Y 446.422,Z 325.875,A -85,B 0,C 180,E1 -8698.7,E2 -8698.7} C_VEL
LIN {X 0,Y 446.463,Z 326,A -85,B 0,C 180,E1 -8699.491,E2 -8699.491} C_VEL
LIN {X 0,Y 450.209,Z 342.936,A -85,B 0,C 180,E1 -8702.28,E2 -8702.28} C_VEL
LIN {X 0,Y 450.452,Z 347.036,A -85,B 0,C 180,E1 -8702.91,E2 -8702.91} C_VEL
LIN {X 0,Y 449.109,Z 371.305,A -85,B 0,C 180,E1 -8706.481,E2 -8706.481} C_VEL
LIN {X 0,Y 447.984,Z 396.334,A -85,B 0,C 180,E1 -8710.115,E2 -8710.115} C_VEL
LIN {X 0,Y 447.357,Z 411.248,A -85,B 0,C 180,E1 -8712.261,E2 -8712.261} C_VEL
LIN {X 0,Y 450.283,Z 438.612,A -85,B 0,C 180,E1 -8712.885,E2 -8712.885} C_VEL
LIN {X 0,Y 449.175,Z 522.189,A -85,B 0,C 180,E1 -8714.429,E2 -8714.429} C_VEL
LIN {X 0,Y 448.668,Z 535.358,A -85,B 0,C 180,E1 -8714.847,E2 -8714.847} C_VEL
LIN {X 0,Y 448.188,Z 547.593,A -85,B 0,C 180,E1 -8715.411,E2 -8715.411} C_VEL
LIN {X 0,Y 447.6,Z 559.463,A -85,B 0,C 180,E1 -8716.146,E2 -8716.146} C_VEL
LIN {X 0,Y 447.054,Z 571.273,A -85,B 0,C 180,E1 -8717.081,E2 -8717.081} C_VEL
LIN {X 0,Y 446.748,Z 580.331,A -85,B 0,C 180,E1 -8717.969,E2 -8717.969} C_VEL
LIN {X 0,Y 446.302,Z 589.931,A -85,B 0,C 180,E1 -8719.107,E2 -8719.107} C_VEL
LIN {X 0,Y 445.944,Z 599.191,A -85,B 0,C 180,E1 -8720.475,E2 -8720.475} C_VEL
LIN {X 0,Y 445.75,Z 606.649,A -85,B 0,C 180,E1 -8721.842,E2 -8721.842} C_VEL
LIN {X 0,Y 445.694,Z 612.595,A -85,B 0,C 180,E1 -8723.208,E2 -8723.208} C_VEL
LIN {X 0,Y 445.655,Z 617.228,A -85,B 0,C 180,E1 -8724.57,E2 -8724.57} C_VEL
LIN {X 0,Y 445.762,Z 619.666,A -85,B 0,C 180,E1 -8725.478,E2 -8725.478} C_VEL
LIN {X 0,Y 445.835,Z 621.642,A -85,B 0,C 180,E1 -8726.385,E2 -8726.385} C_VEL
LIN {X 0,Y 445.73,Z 623.139,A -85,B 0,C 180,E1 -8727.289,E2 -8727.289} C_VEL
LIN {X 0,Y 445.705,Z 624.163,A -85,B 0,C 180,E1 -8728.193,E2 -8728.193} C_VEL
LIN {X 0,Y 445.716,Z 624.77,A -85,B 0,C 180,E1 -8729.096,E2 -8729.096} C_VEL
LIN {X 0,Y 445.743,Z 624.961,A -85,B 0,C 180,E1 -8730,E2 -8730} C_VEL
LIN {X 0,Y 445.725,Z 624.694,A -85,B 0,C 180,E1 -8730.903,E2 -8730.903} C_VEL
LIN {X 0,Y 445.723,Z 623.979,A -85,B 0,C 180,E1 -8731.807,E2 -8731.807} C_VEL
LIN {X 0,Y 445.75,Z 622.85,A -85,B 0,C 180,E1 -8732.711,E2 -8732.711} C_VEL
LIN {X 0,Y 445.815,Z 620.308,A -85,B 0,C 180,E1 -8734.068,E2 -8734.068} C_VEL
LIN {X 0,Y 445.71,Z 616.678,A -85,B 0,C 180,E1 -8735.429,E2 -8735.429} C_VEL
LIN {X 0,Y 445.746,Z 611.872,A -85,B 0,C 180,E1 -8736.801,E2 -8736.801} C_VEL
LIN {X 0,Y 445.838,Z 605.863,A -85,B 0,C 180,E1 -8738.156,E2 -8738.156} C_VEL
LIN {X 0,Y 445.959,Z 598.324,A -85,B 0,C 180,E1 -8739.525,E2 -8739.525} C_VEL
LIN {X 0,Y 446.267,Z 588.937,A -85,B 0,C 180,E1 -8740.893,E2 -8740.893} C_VEL
LIN {X 0,Y 446.646,Z 580.386,A -85,B 0,C 180,E1 -8741.919,E2 -8741.919} C_VEL
LIN {X 0,Y 447.087,Z 569.461,A -85,B 0,C 180,E1 -8743.002,E2 -8743.002} C_VEL
LIN {X 0,Y 447.666,Z 557.164,A -85,B 0,C 180,E1 -8743.968,E2 -8743.968} C_VEL
LIN {X 0,Y 448.407,Z 544.225,A -85,B 0,C 180,E1 -8744.755,E2 -8744.755} C_VEL
LIN {X 0,Y 448.939,Z 531.024,A -85,B 0,C 180,E1 -8745.347,E2 -8745.347} C_VEL
LIN {X 0,Y 449.493,Z 517.402,A -85,B 0,C 180,E1 -8745.763,E2 -8745.763} C_VEL
LIN {X 0,Y 450.539,Z 436.999,A -85,B 0,C 180,E1 -8747.309,E2 -8747.309} C_VEL
LIN {X 0,Y 447.829,Z 410.249,A -85,B 0,C 180,E1 -8747.994,E2 -8747.994} C_VEL
LIN {X 0,Y 447.213,Z 405.286,A -85,B 0,C 180,E1 -8748.156,E2 -8748.156} C_VEL
LIN {X 0,Y 448.042,Z 384.811,A -85,B 0,C 180,E1 -8751.148,E2 -8751.148} C_VEL
LIN {X 0,Y 449.18,Z 362.807,A -85,B 0,C 180,E1 -8754.452,E2 -8754.452} C_VEL
LIN {X 0,Y 450.275,Z 345.351,A -85,B 0,C 180,E1 -8757.168,E2 -8757.168} C_VEL
LIN {X 0,Y 449.858,Z 340.746,A -85,B 0,C 180,E1 -8757.949,E2 -8757.949} C_VEL
LIN {X 0,Y 447.176,Z 328.716,A -85,B 0,C 180,E1 -8760.194,E2 -8760.194} C_VEL
LIN {X 0,Y 446.454,Z 325.879,A -85,B 0,C 180,E1 -8760.771,E2 -8760.771} C_VEL
LIN {X 0,Y 446.448,Z 325.876,A -85,B 0,C 180,E1 -8763.453,E2 -8763.453} C_VEL
LIN {X 0,Y 446.402,Z 325.881,A -85,B 0,C 180,E1 -8766.745,E2 -8766.745} C_VEL
LIN {X 0,Y 446.403,Z 325.88,A -85,B 0,C 180,E1 -8769.516,E2 -8769.516} C_VEL
LIN {X 0,Y 446.39,Z 325.883,A -85,B 0,C 180,E1 -8772.609,E2 -8772.609} C_VEL
LIN {X 0,Y 446.452,Z 325.872,A -85,B 0,C 180,E1 -8775.104,E2 -8775.104} C_VEL
LIN {X 0,Y 446.407,Z 325.879,A -85,B 0,C 180,E1 -8778.606,E2 -8778.606} C_VEL
LIN {X 0,Y 446.4,Z 325.88,A -85,B 0,C 180,E1 -8781.924,E2 -8781.924} C_VEL
LIN {X 0,Y 446.422,Z 325.877,A -85,B 0,C 180,E1 -8785.476,E2 -8785.476} C_VEL
LIN {X 0,Y 446.409,Z 325.877,A -85,B 0,C 180,E1 -8788.699,E2 -8788.699} C_VEL
LIN {X 0,Y 446.425,Z 325.879,A -85,B 0,C 180,E1 -8791.836,E2 -8791.836} C_VEL
LIN {X 0,Y 446.414,Z 325.878,A -85,B 0,C 180,E1 -8794.845,E2 -8794.845} C_VEL
LIN {X 0,Y 446.446,Z 325.876,A -85,B 0,C 180,E1 -8798.246,E2 -8798.246} C_VEL
LIN {X 0,Y 446.421,Z 325.878,A -85,B 0,C 180,E1 -8801.647,E2 -8801.647} C_VEL
LIN {X 0,Y 446.544,Z 326.04,A -85,B 0,C 180,E1 -8804.231,E2 -8804.231} C_VEL
LIN {X 0,Y 451.518,Z 339.156,A -85,B 0,C 180,E1 -8804.786,E2 -8804.786} C_VEL
LIN {X 0,Y 450.127,Z 417.411,A -85,B 0,C 180,E1 -8806.34,E2 -8806.34} C_VEL
LIN {X 0,Y 449.981,Z 430.922,A -85,B 0,C 180,E1 -8806.796,E2 -8806.796} C_VEL
LIN {X 0,Y 449.755,Z 442.693,A -85,B 0,C 180,E1 -8807.363,E2 -8807.363} C_VEL
LIN {X 0,Y 449.431,Z 454.934,A -85,B 0,C 180,E1 -8808.156,E2 -8808.156} C_VEL
LIN {X 0,Y 448.892,Z 465.906,A -85,B 0,C 180,E1 -8809.057,E2 -8809.057} C_VEL
LIN {X 0,Y 448.46,Z 475.78,A -85,B 0,C 180,E1 -8810.073,E2 -8810.073} C_VEL
LIN {X 0,Y 447.941,Z 485.24,A -85,B 0,C 180,E1 -8811.282,E2 -8811.282} C_VEL
LIN {X 0,Y 447.441,Z 493.331,A -85,B 0,C 180,E1 -8812.554,E2 -8812.554} C_VEL
LIN {X 0,Y 447.132,Z 500.212,A -85,B 0,C 180,E1 -8813.909,E2 -8813.909} C_VEL
LIN {X 0,Y 446.789,Z 504.863,A -85,B 0,C 180,E1 -8815.036,E2 -8815.036} C_VEL
LIN {X 0,Y 446.415,Z 509.323,A -85,B 0,C 180,E1 -8816.389,E2 -8816.389} C_VEL
LIN {X 0,Y 446.266,Z 511.643,A -85,B 0,C 180,E1 -8817.292,E2 -8817.292} C_VEL
LIN {X 0,Y 446.297,Z 513.495,A -85,B 0,C 180,E1 -8818.195,E2 -8818.195} C_VEL
LIN {X 0,Y 446.151,Z 514.958,A -85,B 0,C 180,E1 -8819.097,E2 -8819.097} C_VEL
LIN {X 0,Y 446.111,Z 515.952,A -85,B 0,C 180,E1 -8820,E2 -8820} C_VEL
LIN {X 0,Y 446.101,Z 516.527,A -85,B 0,C 180,E1 -8820.902,E2 -8820.902} C_VEL
LIN {X 0,Y 445.883,Z 516.735,A -85,B 0,C 180,E1 -8821.806,E2 -8821.806} C_VEL
LIN {X 0,Y 445.912,Z 516.51,A -85,B 0,C 180,E1 -8822.71,E2 -8822.71} C_VEL
LIN {X 0,Y 445.977,Z 515.833,A -85,B 0,C 180,E1 -8823.614,E2 -8823.614} C_VEL
LIN {X 0,Y 446.104,Z 514.753,A -85,B 0,C 180,E1 -8824.517,E2 -8824.517} C_VEL
LIN {X 0,Y 446.141,Z 513.283,A -85,B 0,C 180,E1 -8825.423,E2 -8825.423} C_VEL
LIN {X 0,Y 446.246,Z 509.743,A -85,B 0,C 180,E1 -8826.956,E2 -8826.956} C_VEL
LIN {X 0,Y 446.404,Z 506.08,A -85,B 0,C 180,E1 -8828.145,E2 -8828.145} C_VEL
LIN {X 0,Y 446.699,Z 499.696,A -85,B 0,C 180,E1 -8829.737,E2 -8829.737} C_VEL
LIN {X 0,Y 447.004,Z 492.727,A -85,B 0,C 180,E1 -8831.104,E2 -8831.104} C_VEL
LIN {X 0,Y 447.36,Z 485.602,A -85,B 0,C 180,E1 -8832.244,E2 -8832.244} C_VEL
LIN {X 0,Y 447.724,Z 476.614,A -85,B 0,C 180,E1 -8833.433,E2 -8833.433} C_VEL
LIN {X 0,Y 448.147,Z 466.323,A -85,B 0,C 180,E1 -8834.531,E2 -8834.531} C_VEL
LIN {X 0,Y 448.54,Z 455.732,A -85,B 0,C 180,E1 -8835.448,E2 -8835.448} C_VEL
LIN {X 0,Y 448.982,Z 444.1,A -85,B 0,C 180,E1 -8836.248,E2 -8836.248} C_VEL
LIN {X 0,Y 449.355,Z 430.782,A -85,B 0,C 180,E1 -8836.935,E2 -8836.935} C_VEL
LIN {X 0,Y 449.463,Z 417.224,A -85,B 0,C 180,E1 -8837.433,E2 -8837.433} C_VEL
LIN {X 0,Y 449.642,Z 399.865,A -85,B 0,C 180,E1 -8837.801,E2 -8837.801} C_VEL
LIN {X 0,Y 450.383,Z 337.487,A -85,B 0,C 180,E1 -8838.936,E2 -8838.936} C_VEL
